# B&R Automation Studio project CleanChemi_SiteManagementSystem (part 2)

### Global.typ - Global data types
```iecst
(*Global Structrues*)
(**)
(*Raw Modbus Data*)

TYPE
	Modbus_Type : 	STRUCT
		Modbus_Alarms : Modbus_Alarm_Type;
		Modbus_Dosing : Modbus_7000_Type;
		Modbus_PeroxyMAX : Modbus_6000_Type;
	END_STRUCT;
END_TYPE

(*Raw Modbus IO*)

TYPE
	Modbus_Alarm_Type : 	STRUCT
		Block48_Int : ARRAY[0..60]OF INT;
	END_STRUCT;
	Modbus_6000_Type : 	STRUCT
		Block1_Int : ARRAY[0..124]OF INT;
		Block2_Int : ARRAY[0..248]OF USINT;
		Block3_Real : ARRAY[0..62]OF REAL;
		Block4_Real : ARRAY[0..62]OF REAL;
		Block5_Real : ARRAY[0..62]OF REAL;
	END_STRUCT;
	Modbus_7000_Type : 	STRUCT
		Block6_Int : ARRAY[0..124]OF INT;
		Block7_Int : ARRAY[0..124]OF INT;
		Block61_Int : ARRAY[0..248]OF USINT;
		Block8_Real : ARRAY[0..62]OF REAL;
		Block9_Real : ARRAY[0..62]OF REAL;
		Block10_Real : ARRAY[0..62]OF REAL;
		Block11_Real : ARRAY[0..62]OF REAL;
	END_STRUCT;
END_TYPE

(**)
(*Final Mapping Variables*)

TYPE
	Skid_type : 	STRUCT
		Pmax_Pump_101 : Pmax_Pump_101_Type;
		Pmax_Pump_101B : Pmax_Pump_101B_Type;
		Pmax_Pump_102 : Pmax_Pump_102_Type;
		Pmax_Pump_103 : Pmax_Pump_103_Type;
		Pmax_Pump_104 : Pmax_Pump_104_Type;
		BufferTank : BufferTank_Variables_Type;
		ConversionRatios : ConversionRatios_Type;
		Sensor_Variables : Sensor_Variables_Type;
		Heartbeat : Heartbeat_Type;
		Status : Status_Type;
		Alarms : Alarms_Type;
		Pmax_General_Variables : Pmax_General_Variables_Type;
		Dosing_Pump_201 : Dosing_Pump_201_Type;
		Dosing_Pump_202 : Dosing_Pump_202_Type;
		Dosing_Pump_203 : Dosing_Pump_203_Type;
		Dosing_Pump_204 : Dosing_Pump_204_Type;
		Dosing_Pump_205 : Dosing_Pump_205_Type;
		Dosing_Pump_206 : Dosing_Pump_206_Type;
		Dosing_Pump_207 : Dosing_Pump_207_Type;
		Dosing_Pump_208 : Dosing_Pump_208_Type;
		VisNum : VisNum_Type;
		VisBool : VisBool_Type;
		ErrorInfo : Skid_ErrorInfo_typ;
		tempAlarm : HA_AlarmX_Core_Buffer_typ;
		Error : BOOL;
		StateResetAlarms : UINT;
		AlarmStartupDelay : TON;
		AlarmXHistory_MpLink : MpComIdentType;
		AlarmX_MpLink : MpComIdentType;
		AlarmCfg : MpAlarmXAlarmConfigType;
		MpAlarmXConfigAlarm : MpAlarmXConfigAlarm;
		i : USINT;
		AlarmName : STRING[80];
		AlarmsInitialized : BOOL;
		Notes : Notes_Type;
		AlarmConfig : AlarmConfig_Type;
		RosterContact : RosterContact_Type;
		UserLock_LastName : STRING[80];
		UserLock_FirstName : STRING[80];
		UserLock : UINT;
	END_STRUCT;
END_TYPE

(**)
(*Alarm Text Messaging Internal CCI Roster*)

TYPE
	RosterContact_Type : 	STRUCT
		Write_Step1 : INT := 0;
		Write_Step2 : INT := 0;
		Write_Step3 : INT := 0;
		Write_Step4 : INT := 0;
		Write_Step5 : INT := 0;
		Write_Step6 : INT := 0;
		Write_Step7 : INT := 0;
		Write_Step8 : INT := 0;
		Contact1_ENABLE : BOOL;
		Contact2_ENABLE : BOOL;
		Contact3_ENABLE : BOOL;
		Contact4_ENABLE : BOOL;
		Contact5_ENABLE : BOOL;
		Contact6_ENABLE : BOOL;
		Contact7_ENABLE : BOOL;
		Contact8_ENABLE : BOOL; (*Pump 202 Visualization Enable Bit 0 = Visible  1 = Hidden*)
		Contact1 : STRING[80];
		Contact2 : STRING[80];
		Contact3 : STRING[80];
		Contact4 : STRING[80];
		Contact5 : STRING[80];
		Contact6 : STRING[80];
		Contact7 : STRING[80];
		Contact8 : STRING[80];
		Phone_Read1 : STRING[10];
		Phone_Read2 : STRING[10];
		Phone_Read3 : STRING[10];
		Phone_Read4 : STRING[10];
		Phone_Read5 : STRING[10];
		Phone_Read6 : STRING[10];
		Phone_Read7 : STRING[10];
		Phone_Read8 : STRING[10];
		Phone_Input1 : STRING[10];
		Phone_Input2 : STRING[10];
		Phone_Input3 : STRING[10];
		Phone_Input4 : STRING[10];
		Phone_Input5 : STRING[10];
		Phone_Input6 : STRING[10];
		Phone_Input7 : STRING[10];
		Phone_Input8 : STRING[10];
	END_STRUCT;
END_TYPE

(*Visualization Components*)

TYPE
	Skid_ErrorInfo_typ : 	STRUCT
		State : STRING[80];
		Text : STRING[255];
		Severity : USINT;
	END_STRUCT;
END_TYPE

(**)

TYPE
	Par_System_type : 	STRUCT
		LanguageCode : STRING[80];
	END_STRUCT;
END_TYPE

(*Retain Machine State After Power Cycle*)

TYPE
	Par_Type : 	STRUCT
		System : Par_System_type;
	END_STRUCT;
END_TYPE

(**)
(*Retain Parameter After Power Cycle*)

TYPE
	Rem_Type : 	STRUCT
		New_Member : USINT;
	END_STRUCT;
END_TYPE

(**)
(*Master Write Command *)

TYPE
	CMD_Type : 	STRUCT
		Stop : BOOL;
		Start : BOOL;
		Write_ESTOP : CMD_Write_ESTOP_Type;
		Write_UNIT_ID : CMD_Write_UNIT_ID_Type;
		Write_UNIT_ACK : CMD_Write_UNIT_ACK_Type;
		Write_P203_STP_CMD : CMD_Write_P203_STP_CMD_Type;
		Write_P203_STRT_CMD : CMD_Write_P203_STRT_CMD_Type;
		Write_P203_HOA : CMD_Write_P203_HOA_Type;
		Write_P203_PPM : CMD_Write_P203_PPM_Type;
		Write_P203_SP : CMD_Write_P203_SP_Type;
		Write_P202_STP_CMD : CMD_Write_P202_STP_CMD_Type;
		Write_P202_STRT_CMD : CMD_Write_P202_STRT_CMD_Type;
		Write_P202_HOA : CMD_Write_P202_HOA_Type;
		Write_P202_PPM : CMD_Write_P202_PPM_Type;
		Write_P202_SP : CMD_Write_P202_SP_Type;
		Write_P104_STP_CMD : CMD_Write_P104_STP_CMD_Type;
		Write_P104_STRT_CMD : CMD_Write_P104_STRT_CMD_Type;
		Write_P104_SP : CMD_Write_P104_SP_Type;
		Write_P103_STP_CMD : CMD_Write_P103_STP_CMD_Type;
		Write_P103_STRT_CMD : CMD_Write_P103_STRT_CMD_Type;
		Write_P103_SP : CMD_Write_P103_SP_Type;
		Write_P102_STP_CMD : CMD_Write_P102_STP_CMD_Type;
		Write_P102_STRT_CMD : CMD_Write_P102_STRT_CMD_Type;
		Write_P102_SP : CMD_Write_P102_SP_Type;
		Write_P101_STP_CMD : CMD_Write_P101_STP_CMD_Type;
		Write_P101_STRT_CMD : CMD_Write_P101_STRT_CMD_Type;
		Write_P101_SP : CMD_Write_P101_SP_Type;
		Write_P201_STP_CMD : CMD_Write_P201_STP_CMD_Type;
		Write_P201_STRT_CMD : CMD_Write_P201_STRT_CMD_Type;
		Write_P201_HOA : CMD_Write_P201_HOA_Type;
		Write_P201_PPM : CMD_Write_P201_PPM_Type;
		Write_P201_SP : CMD_Write_P201_SP_Type;
		Write_EFF_1 : CMD_Write_EFF_1_Type;
		Write_EFF_2 : CMD_Write_EFF_2_Type;
		Write_NAOH_TO_H2O2 : CMD_Write_NAOH_TO_H2O2_Type;
		Write_TRI_TO_H2O2 : CMD_Write_TRI_TO_H2O2_Type;
		Write_PMAX_HOA : CMD_Write_PMAX_HOA_Type;
		Write_PMAX_CONC : CMD_Write_PMAX_CONC_Type;
		Write_HP_CONC : CMD_Write_HP_CONC_Type;
		Write_NAOH_CONC : CMD_Write_NAOH_CONC_Type;
		Write_UNLOCK_CMD : CMD_Write_UNLOCK_CMD_Type;
		Write_LOCK_CMD : CMD_Write_LOCK_CMD_Type;
		Write_FI301_SIM_CMD : CMD_Write_FI301_SIM_CMD_Type;
		Write_FI301_MEA_CMD : CMD_Write_FI301_MEA_CMD_Type;
		Write_FI301_SIM : CMD_Write_FI301_SIM_Type;
		Write_FI302_SIM_CMD : CMD_Write_FI302_SIM_CMD_Type;
		Write_FI302_MEA_CMD : CMD_Write_FI302_MEA_CMD_Type;
		Write_FI302_SIM : CMD_Write_FI302_SIM_Type;
		Write_FI303_SIM_CMD : CMD_Write_FI303_SIM_CMD_Type;
		Write_FI303_MEA_CMD : CMD_Write_FI303_MEA_CMD_Type;
		Write_FI303_SIM : CMD_Write_FI303_SIM_Type;
		Write_XV101_OPEN_CMD : CMD_Write_XV101_OPEN_CMD_Type;
		Write_XV102_OPEN_CMD : CMD_Write_XV102_OPEN_CMD_Type;
		Write_XV103_OPEN_CMD : CMD_Write_XV103_OPEN_CMD_Type;
		Write_XV104_OPEN_CMD : CMD_Write_XV104_OPEN_CMD_Type;
		Write_XV201_OPEN_CMD : CMD_Write_XV201_OPEN_CMD_Type;
		Write_XV202_OPEN_CMD : CMD_Write_XV202_OPEN_CMD_Type;
		Write_XV203_OPEN_CMD : CMD_Write_XV203_OPEN_CMD_Type;
		Write_XV204_OPEN_CMD : CMD_Write_XV204_OPEN_CMD_Type;
		Write_RECALC_CMD : CMD_Write_RECALC_CMD_Type;
		Write_USERADMIN_RESET : CMD_Write_USERADMIN_RESET_Type;
		Write_TOTALIZER_RESET : CMD_Write_TOTALIZER_RESET_Type;
		Write_AS_USER : CMD_Write_AS_USER_Type;
		Write_AS_ACCESS : CMD_Write_AS_ACCESS_Type;
		Write_P204_STP_CMD : CMD_Write_P204_STP_CMD_Type;
		Write_P204_STRT_CMD : CMD_Write_P204_STRT_CMD_Type;
		Write_P204_HOA : CMD_Write_P204_HOA_Type;
		Write_P204_PPM : CMD_Write_P204_PPM_Type;
		Write_P204_SP : CMD_Write_P204_SP_Type;
		Write_FI304_SIM_CMD : CMD_Write_FI304_SIM_CMD_Type;
		Write_FI304_MEA_CMD : CMD_Write_FI304_MEA_CMD_Type;
		Write_FI304_SIM : CMD_Write_FI304_SIM_Type;
		Write_P101_AUTOCAL : CMD_Write_P101_AUTOCAL_Type;
		Write_P101_GAIN : CMD_Write_P101_GAIN_Type;
		Write_P101_STEPADJ : CMD_Write_P101_STEPADJ_Type;
		Write_P101_TOTALADJ : CMD_Write_P101_TOTALADJ_Type;
		Write_P102_AUTOFLO_ADPT : CMD_Write_P102_AUTOFLO_ADPT_Type;
		Write_P102_AUTOCAL : CMD_Write_P102_AUTOCAL_Type;
		Write_P102_GAIN : CMD_Write_P102_GAIN_Type;
		Write_P102_STEPADJ : CMD_Write_P102_STEPADJ_Type;
		Write_P102_TOTALADJ : CMD_Write_P102_TOTALADJ_Type;
		Write_P103_AUTOFLO_ADPT : CMD_Write_P103_AUTOFLO_ADPT_Type;
		Write_P103_AUTOCAL : CMD_Write_P103_AUTOCAL_Type;
		Write_P103_GAIN : CMD_Write_P103_GAIN_Type;
		Write_P103_STEPADJ : CMD_Write_P103_STEPADJ_Type;
		Write_P103_TOTALADJ : CMD_Write_P103_TOTALADJ_Type;
		Write_P104_AUTOFLO_ADPT : CMD_Write_P104_AUTOFLO_ADPT_Type;
		Write_P104_AUTOCAL : CMD_Write_P104_AUTOCAL_Type;
		Write_P104_AUTOCAL_PV : CMD_Write_P104_AUTOCAL_PV_Type;
		Write_P104_GAIN : CMD_Write_P104_GAIN_Type;
		Write_P104_STEPADJ : CMD_Write_P104_STEPADJ_Type;
		Write_P104_TOTALADJ : CMD_Write_P104_TOTALADJ_Type;
		Write_P201_AUTOFLO_ADPT : CMD_Write_P201_AUTOFLO_ADPT_Type;
		Write_P201_AUTOCAL : CMD_Write_P201_AUTOCAL_Type;
		Write_P201_AUTOCAL_PV : CMD_Write_P201_AUTOCAL_PV_Type;
		Write_P201_GAIN : CMD_Write_P201_GAIN_Type;
		Write_P201_STEPADJ : CMD_Write_P201_STEPADJ_Type;
		Write_P201_TOTALADJ : CMD_Write_P201_TOTALADJ_Type;
		Write_P202_AUTOFLO_ADPT : CMD_Write_P202_AUTOFLO_ADPT_Type;
		Write_P202_AUTOCAL : CMD_Write_P202_AUTOCAL_Type;
		Write_P202_AUTOCAL_PV : CMD_Write_P202_AUTOCAL_PV_Type;
		Write_P202_GAIN : CMD_Write_P202_GAIN_Type;
		Write_P202_STEPADJ : CMD_Write_P202_STEPADJ_Type;
		Write_P202_TOTALADJ : CMD_Write_P202_TOTALADJ_Type;
		Write_P203_AUTOFLO_ADPT : CMD_Write_P203_AUTOFLO_ADPT_Type;
		Write_P203_AUTOCAL : CMD_Write_P203_AUTOCAL_Type;
		Write_P203_AUTOCAL_PV : CMD_Write_P203_AUTOCAL_PV_Type;
		Write_P203_GAIN : CMD_Write_P203_GAIN_Type;
		Write_P203_STEPADJ : CMD_Write_P203_STEPADJ_Type;
		Write_P203_TOTALADJ : CMD_Write_P203_TOTALADJ_Type;
		Write_P204_AUTOFLO_ADPT : CMD_Write_P204_AUTOFLO_ADPT_Type;
		Write_P204_AUTOCAL : CMD_Write_P204_AUTOCAL_Type;
		Write_P204_AUTOCAL_PV : CMD_Write_P204_AUTOCAL_PV_Type;
		Write_P204_GAIN : CMD_Write_P204_GAIN_Type;
		Write_P204_STEPADJ : CMD_Write_P204_STEPADJ_Type;
		Write_P204_TOTALADJ : CMD_Write_P204_TOTALADJ_Type;
		Write_PHONE_INPUT1 : CMD_Write_PHONE_INPUT1_Type;
		Write_PHONE_INPUT2 : CMD_Write_PHONE_INPUT2_Type;
		Write_PHONE_INPUT3 : CMD_Write_PHONE_INPUT3_Type;
		Write_PHONE_INPUT4 : CMD_Write_PHONE_INPUT4_Type;
		Write_PHONE_INPUT5 : CMD_Write_PHONE_INPUT5_Type;
		Write_PHONE_INPUT6 : CMD_Write_PHONE_INPUT6_Type;
		Write_PHONE_INPUT7 : CMD_Write_PHONE_INPUT7_Type;
		Write_PHONE_INPUT8 : CMD_Write_PHONE_INPUT8_Type;
		Write_ENABLE_ROSTER1 : CMD_Write_ENABLE_ROSTER1_Type;
		Write_ENABLE_ROSTER2 : CMD_Write_ENABLE_ROSTER2_Type;
		Write_ENABLE_ROSTER3 : CMD_Write_ENABLE_ROSTER3_Type;
		Write_ENABLE_ROSTER4 : CMD_Write_ENABLE_ROSTER4_Type;
		Write_ENABLE_ROSTER5 : CMD_Write_ENABLE_ROSTER5_Type;
		Write_ENABLE_ROSTER6 : CMD_Write_ENABLE_ROSTER6_Type;
		Write_ENABLE_ROSTER7 : CMD_Write_ENABLE_ROSTER7_Type;
		Write_ENABLE_ROSTER8 : CMD_Write_ENABLE_ROSTER8_Type;
		Write_AC_ALARM_ENABLE : CMD_Write_AC_ALARM_ENABLE_Type;
		Write_AC_TXT_ENABLE : CMD_Write_AC_TXT_ENABLE_Type;
		Write_AC_ACTION : CMD_Write_AC_ACTION_Type;
		Write_AC_DELAY : CMD_Write_AC_DELAY_Type;
		Write_AC_OFFSET : CMD_Write_AC_OFFSET_Type;
		Write_AC_THRESHOLD : CMD_Write_AC_THRESHOLD_Type;
	END_STRUCT;
END_TYPE

(**)
(*Misc. Write Commands*)

TYPE
	CMD_Write_ESTOP_Type : 	STRUCT
		wESTOP : UINT := 1;
		Send : BOOL;
	END_STRUCT;
	CMD_Write_UNIT_ACK_Type : 	STRUCT
		wUNIT_ACK : UINT := 1;
	END_STRUCT;
	CMD_Write_AS_ACCESS_Type : 	STRUCT
		Send : BOOL;
		wAS_ACCESS : UINT := 1;
	END_STRUCT;
	CMD_Write_AS_USER_Type : 	STRUCT
		Send : BOOL;
		wAS_USER : UINT := 1;
	END_STRUCT;
	CMD_Write_RECALC_CMD_Type : 	STRUCT
		Send : BOOL;
		wRECALC_CMD : UINT := 1;
	END_STRUCT;
	CMD_Write_USERADMIN_RESET_Type : 	STRUCT
		Send : BOOL;
		wUSERADMIN_RESET : UINT := 1111;
	END_STRUCT;
	CMD_Write_TOTALIZER_RESET_Type : 	STRUCT
		Send : BOOL;
		wTOTALIZER_RESET : UINT := 1;
	END_STRUCT;
	CMD_Write_UNLOCK_CMD_Type : 	STRUCT
		Send : BOOL;
		wUNLOCK_CMD : UINT := 1;
	END_STRUCT;
	CMD_Write_LOCK_CMD_Type : 	STRUCT
		Send : BOOL;
		wLOCK_CMD : UINT := 1;
	END_STRUCT;
	CMD_Write_EFF_1_Type : 	STRUCT
		Send : BOOL;
		wEFF_1 : REAL;
		wEFF_1_SWAPPED : REAL;
	END_STRUCT;
	CMD_Write_EFF_2_Type : 	STRUCT
		Send : BOOL;
		wEFF_2 : REAL;
		wEFF_2_SWAPPED : REAL;
	END_STRUCT;
	CMD_Write_NAOH_TO_H2O2_Type : 	STRUCT
		Send : BOOL;
		wNAOH_TO_H2O2 : REAL;
		wNAOH_TO_H2O2_SWAPPED : REAL;
	END_STRUCT;
	CMD_Write_TRI_TO_H2O2_Type : 	STRUCT
		Send : BOOL;
		wTRI_TO_H2O2 : REAL;
		wTRI_TO_H2O2_SWAPPED : REAL;
	END_STRUCT;
	CMD_Write_PMAX_HOA_Type : 	STRUCT
		Send : BOOL;
		wPMAX_HOA : UINT;
		Cancel : BOOL;
		wPMAX_HOA_String : STRING[80];
	END_STRUCT;
	CMD_Write_PMAX_CONC_Type : 	STRUCT
		Send : BOOL;
		wPMAX_CONC : REAL;
		wPMAX_CONC_SWAPPED : REAL;
	END_STRUCT;
	CMD_Write_HP_CONC_Type : 	STRUCT
		Send : BOOL;
		wHP_CONC : REAL;
		wHP_CONC_SWAPPED : REAL;
	END_STRUCT;
	CMD_Write_NAOH_CONC_Type : 	STRUCT
		Send : BOOL;
		wNAOH_CONC : REAL;
		wNAOH_CONC_SWAPPED : REAL;
	END_STRUCT;
END_TYPE

(*P101 Write Commands*)

TYPE
	CMD_Write_P101_STP_CMD_Type : 	STRUCT
		Send : BOOL;
		wP101_STP_CMD : UINT := 1;
	END_STRUCT;
	CMD_Write_P101_STRT_CMD_Type : 	STRUCT
		Send : BOOL;
		wP101_STRT_CMD : UINT := 1;
	END_STRUCT;
	CMD_Write_P101_SP_Type : 	STRUCT
		Send : BOOL;
		wP101_SP : REAL;
		wP101_SP_SWAPPED : REAL;
	END_STRUCT;
	CMD_Write_P101_AUTOCAL_Type : 	STRUCT
		Send : BOOL;
		wP101_AUTOCAL : UINT := 1;
	END_STRUCT;
	CMD_Write_P101_GAIN_Type : 	STRUCT
		Send : BOOL;
		wP101_GAIN : REAL;
		wP101_GAIN_SWAPPED : REAL;
	END_STRUCT;
	CMD_Write_P101_STEPADJ_Type : 	STRUCT
		Send : BOOL;
		wP101_STEPADJ : REAL;
		wP101_STEPADJ_SWAPPED : REAL;
	END_STRUCT;
	CMD_Write_P101_TOTALADJ_Type : 	STRUCT
		Send : BOOL;
		wP101_TOTALADJ : REAL;
		wP101_TOTALADJ_SWAPPED : REAL;
	END_STRUCT;
END_TYPE

(*P102 Write Commands*)

TYPE
	CMD_Write_P102_STP_CMD_Type : 	STRUCT
		Send : BOOL;
		wP102_STP_CMD : UINT := 1;
	END_STRUCT;
	CMD_Write_P102_STRT_CMD_Type : 	STRUCT
		Send : BOOL;
		wP102_STRT_CMD : UINT := 1;
	END_STRUCT;
	CMD_Write_P102_SP_Type : 	STRUCT
		Send : BOOL;
		wP102_SP : REAL;
		wP102_SP_SWAPPED : REAL;
	END_STRUCT;
	CMD_Write_P102_AUTOFLO_ADPT_Type : 	STRUCT
		Send : BOOL;
		wP102_P102_AUTOFLO_ADPT : UINT := 1;
	END_STRUCT;
	CMD_Write_P102_AUTOCAL_Type : 	STRUCT
		Send : BOOL;
		wP102_AUTOCAL : UINT := 1;
	END_STRUCT;
	CMD_Write_P102_GAIN_Type : 	STRUCT
		Send : BOOL;
		wP102_GAIN : REAL;
		wP102_GAIN_SWAPPED : REAL;
	END_STRUCT;
	CMD_Write_P102_STEPADJ_Type : 	STRUCT
		Send : BOOL;
		wP102_STEPADJ : REAL;
		wP102_STEPADJ_SWAPPED : REAL;
	END_STRUCT;
	CMD_Write_P102_TOTALADJ_Type : 	STRUCT
		Send : BOOL;
		wP102_TOTALADJ : REAL;
		wP102_TOTALADJ_SWAPPED : REAL;
	END_STRUCT;
END_TYPE

(*P103 Write Commands*)

TYPE
	CMD_Write_P103_STP_CMD_Type : 	STRUCT
		Send : BOOL;
		wP103_STP_CMD : UINT := 1;
	END_STRUCT;
	CMD_Write_P103_STRT_CMD_Type : 	STRUCT
		Send : BOOL;
		wP103_STRT_CMD : UINT := 1;
	END_STRUCT;
	CMD_Write_P103_SP_Type : 	STRUCT
		Send : BOOL;
		wP103_SP : REAL;
		wP103_SP_SWAPPED : REAL;
	END_STRUCT;
	CMD_Write_P103_AUTOFLO_ADPT_Type : 	STRUCT
		Send : BOOL;
		wP103_P103_AUTOFLO_ADPT : UINT := 1;
	END_STRUCT;
	CMD_Write_P103_AUTOCAL_Type : 	STRUCT
		Send : BOOL;
		wP103_AUTOCAL : UINT := 1;
	END_STRUCT;
	CMD_Write_P103_GAIN_Type : 	STRUCT
		Send : BOOL;
		wP103_GAIN : REAL;
		wP103_GAIN_SWAPPED : REAL;
	END_STRUCT;
	CMD_Write_P103_STEPADJ_Type : 	STRUCT
		Send : BOOL;
		wP103_STEPADJ : REAL;
		wP103_STEPADJ_SWAPPED : REAL;
	END_STRUCT;
	CMD_Write_P103_TOTALADJ_Type : 	STRUCT
		Send : BOOL;
		wP103_TOTALADJ : REAL;
		wP103_TOTALADJ_SWAPPED : REAL;
	END_STRUCT;
END_TYPE

(*P104 Write Commands*)

TYPE
	CMD_Write_P104_STP_CMD_Type : 	STRUCT
		Send : BOOL;
		wP104_STP_CMD : UINT := 1;
	END_STRUCT;
	CMD_Write_P104_STRT_CMD_Type : 	STRUCT
		Send : BOOL;
		wP104_STRT_CMD : UINT := 1;
	END_STRUCT;
	CMD_Write_P104_SP_Type : 	STRUCT
		Send : BOOL;
		wP104_SP : REAL;
		wP104_SP_SWAPPED : REAL;
	END_STRUCT;
	CMD_Write_P104_AUTOFLO_ADPT_Type : 	STRUCT
		Send : BOOL;
		wP104_P104_AUTOFLO_ADPT : UINT := 1;
	END_STRUCT;
	CMD_Write_P104_AUTOCAL_Type : 	STRUCT
		Send : BOOL;
		wP104_AUTOCAL : UINT := 1;
	END_STRUCT;
	CMD_Write_P104_AUTOCAL_PV_Type : 	STRUCT
		Send : BOOL;
		wP104_AUTOCAL_PV : UINT := 1;
	END_STRUCT;
	CMD_Write_P104_GAIN_Type : 	STRUCT
		Send : BOOL;
		wP104_GAIN : REAL;
		wP104_GAIN_SWAPPED : REAL;
	END_STRUCT;
	CMD_Write_P104_STEPADJ_Type : 	STRUCT
		Send : BOOL;
		wP104_STEPADJ : REAL;
		wP104_STEPADJ_SWAPPED : REAL;
	END_STRUCT;
	CMD_Write_P104_TOTALADJ_Type : 	STRUCT
		Send : BOOL;
		wP104_TOTALADJ : REAL;
		wP104_TOTALADJ_SWAPPED : REAL;
	END_STRUCT;
END_TYPE

(*P201 Write Commands*)

TYPE
	CMD_Write_P201_STP_CMD_Type : 	STRUCT
		Send : BOOL;
		wP201_STP_CMD : UINT := 1;
	END_STRUCT;
	CMD_Write_P201_STRT_CMD_Type : 	STRUCT
		Send : BOOL;
		wP201_STRT_CMD : UINT := 1;
	END_STRUCT;
	CMD_Write_P201_SP_Type : 	STRUCT
		Send : BOOL;
		wP201_SP : REAL;
		wP201_SP_SWAPPED : REAL;
	END_STRUCT;
	CMD_Write_P201_PPM_Type : 	STRUCT
		Send : BOOL;
		wP201_PPM : REAL;
		wP201_PPM_SWAPPED : REAL;
	END_STRUCT;
	CMD_Write_P201_HOA_Type : 	STRUCT
		Cancel : BOOL;
		Send : BOOL;
		wP201_HOA_String : STRING[80];
		wP201_HOA : UINT;
	END_STRUCT;
	CMD_Write_P201_AUTOFLO_ADPT_Type : 	STRUCT
		Send : BOOL;
		wP201_P201_AUTOFLO_ADPT : UINT := 1;
	END_STRUCT;
	CMD_Write_P201_AUTOCAL_Type : 	STRUCT
		Send : BOOL;
		wP201_AUTOCAL : UINT := 1;
	END_STRUCT;
	CMD_Write_P201_AUTOCAL_PV_Type : 	STRUCT
		Send : BOOL;
		wP201_AUTOCAL_PV : UINT := 1;
	END_STRUCT;
	CMD_Write_P201_GAIN_Type : 	STRUCT
		Send : BOOL;
		wP201_GAIN : REAL;
		wP201_GAIN_SWAPPED : REAL;
	END_STRUCT;
	CMD_Write_P201_STEPADJ_Type : 	STRUCT
		Send : BOOL;
		wP201_STEPADJ : REAL;
		wP201_STEPADJ_SWAPPED : REAL;
	END_STRUCT;
	CMD_Write_P201_TOTALADJ_Type : 	STRUCT
		Send : BOOL;
		wP201_TOTALADJ : REAL;
		wP201_TOTALADJ_SWAPPED : REAL;
	END_STRUCT;
END_TYPE

(*P202 Write Commands*)

TYPE
	CMD_Write_P202_STP_CMD_Type : 	STRUCT
		Send : BOOL;
		wP202_STP_CMD : UINT := 1;
	END_STRUCT;
	CMD_Write_P202_STRT_CMD_Type : 	STRUCT
		Send : BOOL;
		wP202_STRT_CMD : UINT := 1;
	END_STRUCT;
	CMD_Write_P202_SP_Type : 	STRUCT
		Send : BOOL;
		wP202_SP : REAL;
		wP202_SP_SWAPPED : REAL;
	END_STRUCT;
	CMD_Write_P202_PPM_Type : 	STRUCT
		Send : BOOL;
		wP202_PPM : REAL;
		wP202_PPM_SWAPPED : REAL;
	END_STRUCT;
	CMD_Write_P202_HOA_Type : 	STRUCT
		Cancel : BOOL;
		Send : BOOL;
		wP202_HOA_String : STRING[80];
		wP202_HOA : UINT;
	END_STRUCT;
	CMD_Write_P202_AUTOFLO_ADPT_Type : 	STRUCT
		Send : BOOL;
		wP202_P202_AUTOFLO_ADPT : UINT := 1;
	END_STRUCT;
	CMD_Write_P202_AUTOCAL_Type : 	STRUCT
		Send : BOOL;
		wP202_AUTOCAL : UINT := 1;
	END_STRUCT;
	CMD_Write_P202_AUTOCAL_PV_Type : 	STRUCT
		Send : BOOL;
		wP202_AUTOCAL_PV : UINT := 1;
	END_STRUCT;
	CMD_Write_P202_GAIN_Type : 	STRUCT
		Send : BOOL;
		wP202_GAIN : REAL;
		wP202_GAIN_SWAPPED : REAL;
	END_STRUCT;
	CMD_Write_P202_STEPADJ_Type : 	STRUCT
		Send : BOOL;
		wP202_STEPADJ : REAL;
		wP202_STEPADJ_SWAPPED : REAL;
	END_STRUCT;
	CMD_Write_P202_TOTALADJ_Type : 	STRUCT
		Send : BOOL;
		wP202_TOTALADJ : REAL;
		wP202_TOTALADJ_SWAPPED : REAL;
	END_STRUCT;
END_TYPE

(*P203 Write Commands*)

TYPE
	CMD_Write_P203_STP_CMD_Type : 	STRUCT
		Send : BOOL;
		wP203_STP_CMD : UINT := 1;
	END_STRUCT;
	CMD_Write_P203_STRT_CMD_Type : 	STRUCT
		Send : BOOL;
		wP203_STRT_CMD : UINT := 1;
	END_STRUCT;
	CMD_Write_P203_SP_Type : 	STRUCT
		Send : BOOL;
		wP203_SP : REAL;
		wP203_SP_SWAPPED : REAL;
	END_STRUCT;
	CMD_Write_P203_PPM_Type : 	STRUCT
		Send : BOOL;
		wP203_PPM : REAL;
		wP203_PPM_SWAPPED : REAL;
	END_STRUCT;
	CMD_Write_P203_HOA_Type : 	STRUCT
		Send : BOOL;
		wP203_HOA : UINT;
		Cancel : BOOL;
		wP203_HOA_String : STRING[80];
	END_STRUCT;
	CMD_Write_P203_AUTOFLO_ADPT_Type : 	STRUCT
		Send : BOOL;
		wP203_P203_AUTOFLO_ADPT : UINT := 1;
	END_STRUCT;
	CMD_Write_P203_AUTOCAL_Type : 	STRUCT
		Send : BOOL;
		wP203_AUTOCAL : UINT := 1;
	END_STRUCT;
	CMD_Write_P203_AUTOCAL_PV_Type : 	STRUCT
		Send : BOOL;
		wP203_AUTOCAL_PV : UINT := 1;
	END_STRUCT;
	CMD_Write_P203_GAIN_Type : 	STRUCT
		Send : BOOL;
		wP203_GAIN : REAL;
		wP203_GAIN_SWAPPED : REAL;
	END_STRUCT;
	CMD_Write_P203_STEPADJ_Type : 	STRUCT
		Send : BOOL;
		wP203_STEPADJ : REAL;
		wP203_STEPADJ_SWAPPED : REAL;
	END_STRUCT;
	CMD_Write_P203_TOTALADJ_Type : 	STRUCT
		Send : BOOL;
		wP203_TOTALADJ : REAL;
		wP203_TOTALADJ_SWAPPED : REAL;
	END_STRUCT;
END_TYPE

(*P204 Write Commands*)

TYPE
	CMD_Write_P204_STP_CMD_Type : 	STRUCT
		Send : BOOL;
		wP204_STP_CMD : UINT := 1;
	END_STRUCT;
	CMD_Write_P204_STRT_CMD_Type : 	STRUCT
		Send : BOOL;
		wP204_STRT_CMD : UINT := 1;
	END_STRUCT;
	CMD_Write_P204_SP_Type : 	STRUCT
		Send : BOOL;
		wP204_SP : REAL;
		wP204_SP_SWAPPED : REAL;
	END_STRUCT;
	CMD_Write_P204_PPM_Type : 	STRUCT
		Send : BOOL;
		wP204_PPM : REAL;
		wP204_PPM_SWAPPED : REAL;
	END_STRUCT;
	CMD_Write_P204_HOA_Type : 	STRUCT
		Send : BOOL;
		wP204_HOA : UINT;
		Cancel : BOOL;
		wP204_HOA_String : STRING[80];
	END_STRUCT;
	CMD_Write_P204_AUTOFLO_ADPT_Type : 	STRUCT
		Send : BOOL;
		wP204_P204_AUTOFLO_ADPT : UINT := 1;
	END_STRUCT;
	CMD_Write_P204_AUTOCAL_Type : 	STRUCT
		Send : BOOL;
		wP204_AUTOCAL : UINT := 1;
	END_STRUCT;
	CMD_Write_P204_AUTOCAL_PV_Type : 	STRUCT
		Send : BOOL;
		wP204_AUTOCAL_PV : UINT := 1;
	END_STRUCT;
	CMD_Write_P204_GAIN_Type : 	STRUCT
		Send : BOOL;
		wP204_GAIN : REAL;
		wP204_GAIN_SWAPPED : REAL;
	END_STRUCT;
	CMD_Write_P204_STEPADJ_Type : 	STRUCT
		Send : BOOL;
		wP204_STEPADJ : REAL;
		wP204_STEPADJ_SWAPPED : REAL;
	END_STRUCT;
	CMD_Write_P204_TOTALADJ_Type : 	STRUCT
		Send : BOOL;
		wP204_TOTALADJ : REAL;
		wP204_TOTALADJ_SWAPPED : REAL;
	END_STRUCT;
END_TYPE

(*UID Write Command*)

TYPE
	CMD_Write_UNIT_ID_Type : 	STRUCT
		Send : BOOL;
		wUNIT_ID : UINT;
	END_STRUCT;
END_TYPE

(*FI301 Write Commands*)

TYPE
	CMD_Write_FI301_SIM_CMD_Type : 	STRUCT
		Send : BOOL;
		wFI301_SIM_CMD : UINT := 1;
	END_STRUCT;
	CMD_Write_FI301_MEA_CMD_Type : 	STRUCT
		Send : BOOL;
		wFI301_MEA_CMD : UINT := 1;
	END_STRUCT;
	CMD_Write_FI301_SIM_Type : 	STRUCT
		Send : BOOL;
		wFI301_SIM : REAL;
		wFI301_SIM_SWAPPED : REAL;
	END_STRUCT;
END_TYPE

(*FI302 Write Commands*)

TYPE
	CMD_Write_FI302_SIM_CMD_Type : 	STRUCT
		Send : BOOL;
		wFI302_SIM_CMD : UINT := 1;
	END_STRUCT;
	CMD_Write_FI302_MEA_CMD_Type : 	STRUCT
		Send : BOOL;
		wFI302_MEA_CMD : UINT := 1;
	END_STRUCT;
	CMD_Write_FI302_SIM_Type : 	STRUCT
		Send : BOOL;
		wFI302_SIM : REAL;
		wFI302_SIM_SWAPPED : REAL;
	END_STRUCT;
END_TYPE

(*FI303 Write Commands*)

TYPE
	CMD_Write_FI303_SIM_CMD_Type : 	STRUCT
		Send : BOOL;
		wFI303_SIM_CMD : UINT := 1;
	END_STRUCT;
	CMD_Write_FI303_MEA_CMD_Type : 	STRUCT
		Send : BOOL;
		wFI303_MEA_CMD : UINT := 1;
	END_STRUCT;
	CMD_Write_FI303_SIM_Type : 	STRUCT
		Send : BOOL;
		wFI303_SIM : REAL;
		wFI303_SIM_SWAPPED : REAL;
	END_STRUCT;
END_TYPE

(*FI304 Write Commands*)

TYPE
	CMD_Write_FI304_SIM_CMD_Type : 	STRUCT
		Send : BOOL;
		wFI304_SIM_CMD : UINT := 1;
	END_STRUCT;
	CMD_Write_FI304_MEA_CMD_Type : 	STRUCT
		Send : BOOL;
		wFI304_MEA_CMD : UINT := 1;
	END_STRUCT;
	CMD_Write_FI304_SIM_Type : 	STRUCT
		Send : BOOL;
		wFI304_SIM : REAL;
		wFI304_SIM_SWAPPED : REAL;
	END_STRUCT;
END_TYPE

(*XV101 Solenoid Commands*)

TYPE
	CMD_Write_XV101_OPEN_CMD_Type : 	STRUCT
		Send : BOOL;
		wXV101_OPEN_CMD : UINT := 1;
	END_STRUCT;
END_TYPE

(*XV102 Solenoid Commands*)

TYPE
	CMD_Write_XV102_OPEN_CMD_Type : 	STRUCT
		Send : BOOL;
		wXV102_OPEN_CMD : UINT := 1;
	END_STRUCT;
END_TYPE

(*XV103 Solenoid Commands*)

TYPE
	CMD_Write_XV103_OPEN_CMD_Type : 	STRUCT
		Send : BOOL;
		wXV103_OPEN_CMD : UINT := 1;
	END_STRUCT;
END_TYPE

(*XV104 Solenoid Commands*)

TYPE
	CMD_Write_XV104_OPEN_CMD_Type : 	STRUCT
		Send : BOOL;
		wXV104_OPEN_CMD : UINT := 1;
	END_STRUCT;
END_TYPE

(*XV201 Solenoid Commands*)

TYPE
	CMD_Write_XV201_OPEN_CMD_Type : 	STRUCT
		Send : BOOL;
		wXV201_OPEN_CMD : UINT := 1;
	END_STRUCT;
END_TYPE

(*XV202 Solenoid Commands*)

TYPE
	CMD_Write_XV202_OPEN_CMD_Type : 	STRUCT
		Send : BOOL;
		wXV202_OPEN_CMD : UINT := 1;
	END_STRUCT;
END_TYPE

(*XV203 Solenoid Commands*)

TYPE
	CMD_Write_XV203_OPEN_CMD_Type : 	STRUCT
		Send : BOOL;
		wXV203_OPEN_CMD : UINT := 1;
	END_STRUCT;
END_TYPE

(*XV204 Solenoid Commands*)

TYPE
	CMD_Write_XV204_OPEN_CMD_Type : 	STRUCT
		Send : BOOL;
		wXV204_OPEN_CMD : UINT := 1;
	END_STRUCT;
END_TYPE

(*Roster Write Commands*)

TYPE
	CMD_Write_PHONE_INPUT1_Type : 	STRUCT
		Send : BOOL;
		wPHONE_INPUT1_ARRAY : ARRAY[0..4]OF UINT;
	END_STRUCT;
	CMD_Write_ENABLE_ROSTER1_Type : 	STRUCT
		Send : BOOL;
		wENABLE_ROSTER1 : UINT := 0;
	END_STRUCT;
	CMD_Write_PHONE_INPUT2_Type : 	STRUCT
		Send : BOOL;
		wPHONE_INPUT2_ARRAY : ARRAY[0..4]OF UINT;
	END_STRUCT;
	CMD_Write_ENABLE_ROSTER2_Type : 	STRUCT
		Send : BOOL;
		wENABLE_ROSTER2 : UINT := 0;
	END_STRUCT;
	CMD_Write_PHONE_INPUT3_Type : 	STRUCT
		Send : BOOL;
		wPHONE_INPUT3_ARRAY : ARRAY[0..4]OF UINT;
	END_STRUCT;
	CMD_Write_ENABLE_ROSTER3_Type : 	STRUCT
		Send : BOOL;
		wENABLE_ROSTER3 : UINT := 0;
	END_STRUCT;
	CMD_Write_PHONE_INPUT4_Type : 	STRUCT
		Send : BOOL;
		wPHONE_INPUT4_ARRAY : ARRAY[0..4]OF UINT;
	END_STRUCT;
	CMD_Write_ENABLE_ROSTER4_Type : 	STRUCT
		Send : BOOL;
		wENABLE_ROSTER4 : UINT := 0;
	END_STRUCT;
	CMD_Write_PHONE_INPUT5_Type : 	STRUCT
		Send : BOOL;
		wPHONE_INPUT5_ARRAY : ARRAY[0..4]OF UINT;
	END_STRUCT;
	CMD_Write_ENABLE_ROSTER5_Type : 	STRUCT
		Send : BOOL;
		wENABLE_ROSTER5 : UINT := 0;
	END_STRUCT;
	CMD_Write_PHONE_INPUT6_Type : 	STRUCT
		Send : BOOL;
		wPHONE_INPUT6_ARRAY : ARRAY[0..4]OF UINT;
	END_STRUCT;
	CMD_Write_ENABLE_ROSTER6_Type : 	STRUCT
		Send : BOOL;
		wENABLE_ROSTER6 : UINT := 0;
	END_STRUCT;
	CMD_Write_PHONE_INPUT7_Type : 	STRUCT
		Send : BOOL;
		wPHONE_INPUT7_ARRAY : ARRAY[0..4]OF UINT;
	END_STRUCT;
	CMD_Write_ENABLE_ROSTER7_Type : 	STRUCT
		Send : BOOL;
		wENABLE_ROSTER7 : UINT := 0;
	END_STRUCT;
	CMD_Write_PHONE_INPUT8_Type : 	STRUCT
		Send : BOOL;
		wPHONE_INPUT8_ARRAY : ARRAY[0..4]OF UINT;
	END_STRUCT;
	CMD_Write_ENABLE_ROSTER8_Type : 	STRUCT
		Send : BOOL;
		wENABLE_ROSTER8 : UINT := 0;
	END_STRUCT;
END_TYPE

(*Alarm Configuration Write Commands*)

TYPE
	CMD_Write_AC_ALARM_ENABLE_Type : 	STRUCT
		Send : BOOL;
		wAC_ALARM_ENABLE : UINT := 0;
	END_STRUCT;
	CMD_Write_AC_TXT_ENABLE_Type : 	STRUCT
		Send : BOOL;
		wAC_TXT_ENABLE : UINT := 0;
	END_STRUCT;
	CMD_Write_AC_ACTION_Type : 	STRUCT
		Send : BOOL;
		wAC_ACTION : UINT := 0;
	END_STRUCT;
	CMD_Write_AC_DELAY_Type : 	STRUCT
		Send : BOOL;
		wAC_DELAY : UDINT := 0;
	END_STRUCT;
	CMD_Write_AC_OFFSET_Type : 	STRUCT
		Send : BOOL;
		wAC_OFFSET : UINT := 0;
	END_STRUCT;
	CMD_Write_AC_THRESHOLD_Type : 	STRUCT
		Send : BOOL;
		wAC_THRESHOLD : REAL;
		wAC_THRESHOLD_SWAPPED : REAL;
	END_STRUCT;
END_TYPE

(**)

TYPE
	Vis_Type : 	STRUCT
		Pumps : USINT;
		Main : Vis_Main_Type;
		Global : Vis_Global;
		Alarms_HR : ARRAY[0..MAX_SKIDS_HR]OF Vis_Alarms_Type;
		Alarms_LR : ARRAY[0..MAX_SKIDS_LR]OF Vis_Alarms_Type;
		Alarms_Global : Vis_Alarms_Type;
		Process : Vis_Process_Type;
	END_STRUCT;
	Vis_Global : 	STRUCT
		ClientInfo : ARRAY[0..MAX_CLIENTS]OF Vis_Global_ClientInfo;
		ErrorReset : BOOL;
	END_STRUCT;
	Vis_Global_ClientInfo : 	STRUCT
		LoginFailed : BOOL;
		LogoutSuccess : BOOL;
		LoginSuccess : BOOL;
		LogoutRequest : BOOL;
		LoginRequest : BOOL;
		Password : STRING[80];
		User : STRING[80];
		SelectedSkidIdx : USINT;
		UserID : STRING[80];
		IsValid : BOOL;
		LoginBypass : BOOL;
		LoginErrorInfo : STRING[80];
		SelectedAlrm_UnitID : STRING[80];
		SelectedAlrm_Skid : STRING[80];
		GoToSkid : BOOL;
		SelectedAlrmIndx_Temp : UINT;
		SelectedAlrmIndx : UINT;
		API_FIRST_NAME : STRING[80];
		API_LAST_NAME : STRING[80];
		API_ID : UINT;
	END_STRUCT;
	Vis_Alarms_Type : 	STRUCT
		Active : Vis_Alarms_Active_typ;
		History : Vis_Alarms_History_typ;
	END_STRUCT;
	Vis_Alarms_Active_typ : 	STRUCT
		UIConnect : MpAlarmXListUIConnectType;
		Reset : BOOL;
		PageDown : BOOL;
		PageUp : BOOL;
		SelectedIndex_Temp : UINT;
		SelectedIndex : UINT;
		TableConfig : STRING[255];
		TempINT : INT;
		TempSTRING : STRING[30];
		Enable : BOOL;
		Visable : BOOL;
		AckAll : BOOL;
	END_STRUCT;
	Vis_Alarms_History_typ : 	STRUCT
		UIConnect : MpAlarmXHistoryUIConnectType;
		State : ARRAY[0..49]OF UINT;
		Clear : BOOL;
		PageDown : BOOL;
		PageUp : BOOL;
		Export : BOOL;
		SelectedIndex : UINT;
		TableConfig : STRING[255];
		TempINT : INT;
		TempSTRING : STRING[30];
	END_STRUCT;
	Vis_Main_Internal_Type : 	STRUCT
		IP_WSTRING_Temp : WSTRING[80];
		SkidAlarmName : STRING[80];
	END_STRUCT;
	Vis_Main_Out_Type : 	STRUCT
		IPAddressDataProv_HR : ARRAY[0..MAX_SKIDS_HR]OF WSTRING[80];
		IPAddressDataProv_LR : ARRAY[0..MAX_SKIDS_LR]OF WSTRING[80];
		DialogOpen : BOOL;
		SkidIPAddress_LR : ARRAY[0..MAX_SKIDS_LR]OF STRING[20];
		SkidIPAddress_HR : ARRAY[0..MAX_SKIDS_HR]OF STRING[20];
	END_STRUCT;
	Vis_Main_In_Type : 	STRUCT
		SelectedSkidSessionVar : INT;
		AckAllAlarms_Skid_HR : ARRAY[0..100]OF BOOL;
		AckAllAlarms_Skid_LR : ARRAY[0..100]OF BOOL;
	END_STRUCT;
	Vis_Process_Internal_Type : 	STRUCT
		In : Vis_Main_In_Type;
		Internal : Vis_Main_Internal_Type;
		Out : Vis_Main_Out_Type;
	END_STRUCT;
	Vis_Process_Out_ST_Type : 	STRUCT
		PI101_Indicator : STRING[80];
		PI101_Gauge : REAL;
		CD101_Indicator : STRING[80];
		CD101_Gauge : REAL;
		CD102_Indicator : STRING[80];
		CD102_Gauge : REAL;
		GEN_Indicator : STRING[80];
		UNIT_Indicator : STRING[80];
		P201_Indicator : STRING[80];
		P202_Indicator : STRING[80];
		P203_Indicator : STRING[80];
		FI_PlantFlowCombined : REAL;
		UnitNumber : STRING[80];
	END_STRUCT;
	Vis_Process_Out_Type : 	STRUCT
		SummaryTiles : ARRAY[0..MAX_SKIDS_LR]OF Vis_Process_Out_ST_Type;
	END_STRUCT;
	Vis_Process_In_Type : 	STRUCT
		In : Vis_Main_In_Type;
		Internal : Vis_Main_Internal_Type;
		Out : Vis_Main_Out_Type;
	END_STRUCT;
	Vis_Process_Type : 	STRUCT
		In : Vis_Process_In_Type;
		Internal : Vis_Process_Internal_Type;
		Out : Vis_Process_Out_Type;
	END_STRUCT;
	Vis_Main_Type : 	STRUCT
		In : Vis_Main_In_Type;
		Internal : Vis_Main_Internal_Type;
		Out : Vis_Main_Out_Type;
	END_STRUCT;
END_TYPE

(*Bool Toggles for Hiding Visualiazation Elements*)

TYPE
	VisBool_Type : 	STRUCT
		P104_PV_FIT_EN : BOOL;
		P104_PV_PFIT_EN : BOOL;
		P201_PV_FIT_EN : BOOL;
		P201_PV_PFIT_EN : BOOL;
		P202_PV_FIT_EN : BOOL;
		P202_PV_PFIT_EN : BOOL;
		P203_PV_FIT_EN : BOOL;
		P203_PV_PFIT_EN : BOOL;
		P104_PV_FIT : BOOL;
		P104_PV_PFIT : BOOL;
		P201_PV_FIT : BOOL;
		P201_PV_PFIT : BOOL;
		P202_PV_FIT : BOOL;
		P202_PV_PFIT : BOOL;
		P203_PV_FIT : BOOL;
		P203_PV_PFIT : BOOL;
		P102_AUTOFLOW_ON_EN : BOOL;
		P102_AUTOFLOW_OFF_EN : BOOL;
		P103_AUTOFLOW_ON_EN : BOOL;
		P103_AUTOFLOW_OFF_EN : BOOL;
		P104_AUTOFLOW_ON_EN : BOOL;
		P104_AUTOFLOW_OFF_EN : BOOL;
		P201_AUTOFLOW_ON_EN : BOOL;
		P201_AUTOFLOW_OFF_EN : BOOL;
		P202_AUTOFLOW_ON_EN : BOOL;
		P202_AUTOFLOW_OFF_EN : BOOL;
		P203_AUTOFLOW_ON_EN : BOOL;
		P203_AUTOFLOW_OFF_EN : BOOL;
		P102_AUTOFLOW_ON : BOOL;
		P102_AUTOFLOW_OFF : BOOL;
		P103_AUTOFLOW_ON : BOOL;
		P103_AUTOFLOW_OFF : BOOL;
		P104_AUTOFLOW_ON : BOOL;
		P104_AUTOFLOW_OFF : BOOL;
		P201_AUTOFLOW_ON : BOOL;
		P201_AUTOFLOW_OFF : BOOL;
		P202_AUTOFLOW_ON : BOOL;
		P202_AUTOFLOW_OFF : BOOL;
		P203_AUTOFLOW_ON : BOOL;
		P203_AUTOFLOW_OFF : BOOL;
		P101_AUTOCAL_ON_EN : BOOL;
		P101_AUTOCAL_OFF_EN : BOOL;
		P102_AUTOCAL_ON_EN : BOOL;
		P102_AUTOCAL_OFF_EN : BOOL;
		P103_AUTOCAL_ON_EN : BOOL;
		P103_AUTOCAL_OFF_EN : BOOL;
		P104_AUTOCAL_ON_EN : BOOL;
		P104_AUTOCAL_OFF_EN : BOOL;
		P201_AUTOCAL_ON_EN : BOOL;
		P201_AUTOCAL_OFF_EN : BOOL;
		P202_AUTOCAL_ON_EN : BOOL;
		P202_AUTOCAL_OFF_EN : BOOL;
		P203_AUTOCAL_ON_EN : BOOL;
		P203_AUTOCAL_OFF_EN : BOOL;
		P101_AUTOCAL_ON : BOOL;
		P101_AUTOCAL_OFF : BOOL;
		P102_AUTOCAL_ON : BOOL;
		P102_AUTOCAL_OFF : BOOL;
		P103_AUTOCAL_ON : BOOL;
		P103_AUTOCAL_OFF : BOOL;
		P104_AUTOCAL_ON : BOOL;
		P104_AUTOCAL_OFF : BOOL;
		P201_AUTOCAL_ON : BOOL;
		P201_AUTOCAL_OFF : BOOL;
		P202_AUTOCAL_ON : BOOL;
		P202_AUTOCAL_OFF : BOOL;
		P203_AUTOCAL_ON : BOOL;
		P203_AUTOCAL_OFF : BOOL;
		P204_WARN : BOOL;
		P204_ALARM : BOOL;
		P203_WARN : BOOL;
		P203_ALARM : BOOL;
		P202_WARN : BOOL;
		P202_ALARM : BOOL;
		P201_WARN : BOOL;
		P201_ALARM : BOOL;
		P102_WARN : BOOL;
		P102_ALARM : BOOL;
		P103_WARN : BOOL;
		P103_ALARM : BOOL;
		P104_WARN : BOOL;
		P104_ALARM : BOOL;
		P102_LS : BOOL;
		P103_LS : BOOL;
		LSHH200 : BOOL;
		P204_ENABLE_OPP : BOOL;
		P203_ENABLE_OPP : BOOL;
		P202_ENABLE_OPP : BOOL;
		P201_ENABLE_OPP : BOOL;
		P201_SP : BOOL;
		P202_SP : BOOL;
		P203_SP : BOOL;
		P204_SP : BOOL;
		P201_PPM : BOOL;
		P202_PPM : BOOL;
		P203_PPM : BOOL;
		P204_PPM : BOOL;
		PMAX_MANUAL : BOOL;
		P101_DMEYELLOW : BOOL;
		P101_DMEGREEN : BOOL;
		P102_DDAGREEN : BOOL;
		P103_DDAGREEN : BOOL;
		P104_DDAGREEN : BOOL;
		P202_DDAGREEN : BOOL;
		P203_DDAGREEN : BOOL;
		P102_DDAYELLOW : BOOL;
		P103_DDAYELLOW : BOOL;
		P104_DDAYELLOW : BOOL;
		P201_DDAYELLOW : BOOL;
		P202_DDAYELLOW : BOOL;
		P203_DDAYELLOW : BOOL;
		P201_DDAGREEN : BOOL;
		P201_DDA : BOOL;
		P201_DMEYELLOW : BOOL;
		P201_DMEGREEN : BOOL;
		P201_DME : BOOL;
		P201_APPM : BOOL;
		P202_APPM : BOOL;
		P203_APPM : BOOL;
		P204_APPM : BOOL;
		FI304_MODE : BOOL;
		FI303_MODE : BOOL;
		FI302_MODE : BOOL;
		FI301_MODE : BOOL;
		FI301_MODE_OPP : BOOL;
		FI302_MODE_OPP : BOOL;
		FI303_MODE_OPP : BOOL;
		FI304_MODE_OPP : BOOL;
		XV101 : BOOL;
		XV102 : BOOL;
		XV104 : BOOL;
		XV101_ERROR : BOOL;
		XV101_OPP : BOOL;
		XV102_OPP : BOOL;
		XV103_OPP : BOOL;
		XV104_OPP : BOOL;
		XV201_OPP : BOOL;
		XV202_OPP : BOOL;
		XV203_OPP : BOOL;
		XV204_OPP : BOOL;
		P201_PTYPE_OPP : BOOL;
		P101_MODE : BOOL;
		P102_MODE : BOOL;
		P103_MODE : BOOL;
		P104_MODE : BOOL;
		P201_MODE : BOOL;
		P202_MODE : BOOL;
		P203_MODE : BOOL;
		P204_MODE : BOOL;
		HR_TYPE : BOOL;
		LR_TYPE : BOOL;
		HEARTBEAT : BOOL;
		IOSTATUS : BOOL;
		CD102_TARGETHI : REAL;
		CD102_TARGETLO : REAL;
		CD101_TARGETHI : REAL;
		CD101_TARGETLO : REAL;
		ROSTER1_DISABLE : BOOL;
		ROSTER1_ENABLE : BOOL;
		ROSTER2_DISABLE : BOOL;
		ROSTER2_ENABLE : BOOL;
		ROSTER3_DISABLE : BOOL;
		ROSTER3_ENABLE : BOOL;
		ROSTER4_DISABLE : BOOL;
		ROSTER4_ENABLE : BOOL;
		ROSTER5_DISABLE : BOOL;
		ROSTER5_ENABLE : BOOL;
		ROSTER6_DISABLE : BOOL;
		ROSTER6_ENABLE : BOOL;
		ROSTER7_DISABLE : BOOL;
		ROSTER7_ENABLE : BOOL;
		ROSTER8_DISABLE : BOOL;
		ROSTER8_ENABLE : BOOL;
		ROSTER1_DIS : BOOL;
		ROSTER1_EN : BOOL;
		ROSTER2_DIS : BOOL;
		ROSTER2_EN : BOOL;
		ROSTER3_DIS : BOOL;
		ROSTER3_EN : BOOL;
		ROSTER4_DIS : BOOL;
		ROSTER4_EN : BOOL;
		ROSTER5_DIS : BOOL;
		ROSTER5_EN : BOOL;
		ROSTER6_DIS : BOOL;
		ROSTER6_EN : BOOL;
		ROSTER7_DIS : BOOL;
		ROSTER7_EN : BOOL;
		ROSTER8_DIS : BOOL;
		ROSTER8_EN : BOOL;
		SEND_ROSTER1 : BOOL;
		SEND_ROSTER2 : BOOL;
		SEND_ROSTER3 : BOOL;
		SEND_ROSTER4 : BOOL;
		SEND_ROSTER5 : BOOL;
		SEND_ROSTER6 : BOOL;
		SEND_ROSTER7 : BOOL;
		SEND_ROSTER8 : BOOL;
	END_STRUCT;
	VisNum_Type : 	STRUCT
		P101_TOTALADJ_IN : REAL;
		P102_TOTALADJ_IN : REAL;
		P103_TOTALADJ_IN : REAL;
		P104_TOTALADJ_IN : REAL;
		P201_TOTALADJ_IN : REAL;
		P202_TOTALADJ_IN : REAL;
		P203_TOTALADJ_IN : REAL;
		P101_TOTALADJ : REAL;
		P102_TOTALADJ : REAL;
		P103_TOTALADJ : REAL;
		P104_TOTALADJ : REAL;
		P201_TOTALADJ : REAL;
		P202_TOTALADJ : REAL;
		P203_TOTALADJ : REAL;
		P101_STEPADJ_IN : REAL;
		P102_STEPADJ_IN : REAL;
		P103_STEPADJ_IN : REAL;
		P104_STEPADJ_IN : REAL;
		P201_STEPADJ_IN : REAL;
		P202_STEPADJ_IN : REAL;
		P203_STEPADJ_IN : REAL;
		P101_STEPADJ : REAL;
		P102_STEPADJ : REAL;
		P103_STEPADJ : REAL;
		P104_STEPADJ : REAL;
		P201_STEPADJ : REAL;
		P202_STEPADJ : REAL;
		P203_STEPADJ : REAL;
		P101_GAIN : REAL;
		P102_GAIN : REAL;
		P103_GAIN : REAL;
		P104_GAIN : REAL;
		P201_GAIN : REAL;
		P202_GAIN : REAL;
		P203_GAIN : REAL;
		P101_GAIN_IN : REAL;
		P102_GAIN_IN : REAL;
		P103_GAIN_IN : REAL;
		P104_GAIN_IN : REAL;
		P201_GAIN_IN : REAL;
		P202_GAIN_IN : REAL;
		P203_GAIN_IN : REAL;
	END_STRUCT;
END_TYPE

(**)

TYPE
	Recipe_type : 	STRUCT
		Contacts : RosterContact_Type;
		Notes : STRING[80];
	END_STRUCT;
	Notes_Type : 	STRUCT
		LOCATION : STRING[80];
	END_STRUCT;
END_TYPE

(**)
(*Sensors, Flowmeters, Solenoids Variables*)

TYPE
	Sensor_Variables_Type : 	STRUCT  (*Flowmeter and Other Misc Sensor Variables*)
		WASTE_LVL : BOOL; (*Waste Container Level Full Indicator*)
		SERNSORS_CONFIG : UINT; (*Datamap for sensors: DCBA >> sensor301 is type A, sensor302 is type B, sensor303 is type C, sensor304 is type D*)
		SENSOR301 : REAL; (*Sensor 301 Reading*)
		SENSOR302 : REAL; (*Sensor 302 Reading*)
		SENSOR303 : REAL; (*Sensor 303 Reading*)
		SENSOR304 : REAL; (*Sensor 304 Reading*)
		FI301 : REAL; (*Flowmeter 1 Reading*)
		FI301_QT : REAL; (*Totalized Flowmeter 1*)
		FI301_MODE : UINT; (*FI301 Mode 0 = Measure  1 = Simulation*)
		FI302 : REAL; (*Flowmeter 2 Reading*)
		FI302_QT : REAL; (*Totalized Flowmeter 2*)
		FI302_MODE : UINT; (*FI302 Mode 0 = Measure  1 = Simulation*)
		FI303 : REAL; (*Flowmeter 3 Reading*)
		FI303_QT : REAL; (*Totalized Flowmeter 3*)
		FI303_MODE : UINT; (*FI303 Mode 0 = Measure  1 = Simulation*)
		FI304 : REAL; (*Flowmeter 4 Reading*)
		FI304_QT : REAL; (*Totalized Flowmeter 4*)
		FI304_MODE : UINT; (*FI304 Mode 0 = Measure  1 = Simulation*)
		CD101 : REAL; (*Current Transducer 101*)
		CD101_SP : REAL; (*Current Transducer 101 Setpoint*)
		CD102 : REAL; (*Current Transducer 102*)
		CD102_SP : REAL; (*Current Transducer 102 Setpoint*)
		CD103 : REAL; (*Current Transducer 103*)
		CD103_SP : REAL; (*Current Transducer 103 Setpoint*)
		CD101_TI : REAL; (*Temperature After Caustic*)
		CD102_TI : REAL; (*Temperature After Hydrogen Peroxide*)
		CD103_TI : REAL; (*Temperature After Hydrogen Peroxide*)
		XV101_ENABLE : UINT; (*P101 Suction Side Solenoid Feedback Installed on Skid (0 = not installed 1 = installed)*)
		XV101 : UINT; (*P101 Suction Side Solenoid Feedback*)
		XV102 : UINT; (*P102 Off Gas Solenoid Valve*)
		XV103 : UINT; (*P103 Off Gas Solenoid Valve*)
		XV104 : UINT; (*P104 Off Gas Solenoid Valve*)
		XV201 : UINT; (*P201 Off Gas Solenoid Valve*)
		XV202 : UINT; (*P202 Off Gas Solenoid Valve*)
		XV203 : UINT; (*P203 Off Gas Solenoid Valve*)
		XV204 : UINT; (*P204 Off Gas Solenoid Valve*)
	END_STRUCT;
END_TYPE

(**)
(*Alarms*)

TYPE
	AlarmConfig_Type : 	STRUCT  (*Alarm Configuration Parameters*)
		wAC_ALARM_ENABLE_ADDR : UINT; (*Alarm Enable Status Register Address*)
		AC_ENABLE : UINT; (*Alarm and Text Enable Status*)
		AC_ALARM_ENABLE : STRING[10]; (*Alarm Enable Status*)
		wAC_TXT_ENABLE_ADDR : UINT; (*Text alerts enabled Register Address*)
		AC_TXT_ENABLE : STRING[10]; (*Text alerts enabled*)
		AC_LR_ENABLE : BOOL; (*Alarm exists on Low Rate*)
		AC_HR_ENABLE : BOOL; (*Alarm exists on High Rate*)
		AC_ACTION_ENABLE : BOOL; (*Action present and associated with alarm*)
		AC_DESCRIPTION : STRING[40]; (*Description of Alarm*)
		AC_THRESHOLD_UNIT : STRING[10]; (*Units for alarm threshold*)
		wAC_ACTION_ADDR : UINT; (*Alarm action Register Address*)
		AC_ACTION : UINT; (*Alarm action*)
		wAC_DELAY_ADDR : UINT; (*Time delay on alarming Register Address*)
		AC_DELAY : UINT; (*Time delay on alarming*)
		AC_OFFSET : UINT; (*Offset for reference to alarms list for PLC *)
		wAC_THRESHOLD_ADDR : UINT; (*Alarm threshold value Register Address*)
		AC_THRESHOLD : REAL; (*Alarm threshold value*)
	END_STRUCT;
	Alarms_Type : 	STRUCT  (*General Alarm Variables*)
		ALARM_AB1 : INT; (*General Alarm Block 1*)
		ALARM_AB2 : INT; (*General Alarm Block 2*)
		ALARM_AB3 : INT; (*General Alarm Block 3*)
		ALARM_AB4 : INT; (*General Alarm Block 4*)
		ALARM_AB5 : INT; (*General Alarm Block 5*)
		ALARM_AB6 : INT; (*General Alarm Block 6*)
		ALARM_AB7 : INT; (*General Alarm Block 7*)
		ALARM_AB8 : INT; (*General Alarm Block 8*)
		ALARM_AB9 : INT; (*General Alarm Block 9*)
		ALARM_AB10 : INT; (*General Alarm Block 10*)
		ALARM_AB11 : INT; (*General Alarm Block 11*)
		ALARM_AB12 : INT; (*General Alarm Block 12*)
		ALARM_AB13 : INT; (*General Alarm Block 13*)
		ALARM_AB14 : INT; (*General Alarm Block 14*)
		ALARM_AB15 : INT; (*General Alarm Block 15*)
		ALARM_AB16 : INT; (*General Alarm Block 16*)
		ALARM_AB17 : INT; (*General Alarm Block 17*)
		ALARM_AB18 : INT; (*General Alarm Block 18*)
		ALARM_AB19 : INT; (*General Alarm Block 19*)
	END_STRUCT;
END_TYPE

(*Status*)

TYPE
	Status_Type : 	STRUCT  (*General Alarm Variables*)
		P201_STATUS : STRING[20]; (*P201 pump status*)
		P202_STATUS : STRING[20]; (*P202 pump status*)
		P203_STATUS : STRING[20]; (*P203 pump status*)
		PMAX_HOA : STRING[20]; (*Pmax HOA  status*)
		PMAX_STATUS : STRING[20]; (*Pmax unit status*)
	END_STRUCT;
END_TYPE

(**)
(*Heartbeat*)

TYPE
	Heartbeat_Type : 	STRUCT  (*Heartbeat Connection Status Components*)
		PREVIOUS_HEARTBEAT : INT; (*Last value of heartbeat from PLC*)
		MODBUS_RESET : R_TRIG; (*Timer window to detect heartbeat*)
		UNCHANGED_TIMER : TON; (*Timer window to detect heartbeat*)
		SYSTEM_OFFLINE : BOOL; (*System Online Status (1=Offline)*)
	END_STRUCT;
END_TYPE

(**)
(*Conversion/Chem Reaction Efficiencies*)

TYPE
	ConversionRatios_Type : 	STRUCT  (*Efficiency Conversion Ratio Variables*)
		EFF_1 : REAL; (*HP to PAA Conversion Efficiency *)
		EFF_2 : REAL; (*Acetyl Conversion Efficiency *)
		TRI_TO_H2O2 : REAL; (*Molar Ratio of Triacetin to HP*)
		NAOH_TO_TRI : REAL; (*Molar Ratio of NaOH to TRI*)
		NAOH_TO_H2O2 : REAL; (*Molar Ratio of NaOH to HP*)
	END_STRUCT;
END_TYPE

(**)
(*Pmax Generation General Variables*)

TYPE
	Pmax_General_Variables_Type : 	STRUCT  (*PeroxyMax General Variables*)
		PLC_REV_A : REAL; (*PLC Revision Part A*)
		PLC_REV_B : REAL; (*PLC Revision Part B*)
		HMI_REV_A : REAL; (*HMI Revision Part A*)
		HMI_REV_B : REAL; (*HMI Revision Part B*)
		SCREEN_LOCK : BOOL; (*Unit HMI Lockout from SCADA, 1 = Locked   0 = Unlocked*)
		UNIT_ID : UINT; (*Pmax Skid ID*)
		PMAX_HOA : UINT; (*Pmax Generation is ON*)
		PMAX_STATUS : UINT; (*Pmax Status*)
		PMAX_CONC : REAL; (*Pmax Concentration*)
		PMAX_PV : REAL; (*Pmax Present Value*)
		PMAX_RATE : REAL; (*Pmax Rate*)
		HP_CONC_OD : REAL; (*HP Concentration On Deck*)
		HP_CONC : REAL; (*HP Concentration*)
		NAOH_CONC_OD : REAL; (*NaOh Concentration On Deck*)
		NAOH_CONC : REAL; (*NaOh Concentration*)
		USER_ID : UINT; (*Current Local User*)
		USER_ACCESS : UINT; (*Current Local User Access Level*)
		UNIT_TYPE : UINT; (*Unit Type ()*)
		UNIT_ID_DOSE : UINT;
		HEARTBEAT : INT; (*Unit Heartbeat*)
	END_STRUCT;
END_TYPE

(**)
(*Buffer Tank*)

TYPE
	BufferTank_Variables_Type : 	STRUCT  (*Buffer Tank Variables*)
		LSHH200 : REAL; (*Buffer Tank High High Sensor*)
		LI200P : REAL; (*Buffer Tank Level Percent*)
		LI200 : REAL; (*Buffer Tank Level*)
		DRAINTIME_SP : REAL; (*Tank Draintime Setpoint*)
		DRAINTIME_PV : REAL; (*Tank Draintime Present Value*)
		FILLTIME_SP : REAL; (*Tank Filltime Setpoint*)
		FILLTIME_PV : REAL; (*Tank Filltime Present Value*)
		BT_PERCENT : REAL; (*Buffer Tank Fill Percent*)
	END_STRUCT;
END_TYPE

(**)
(*PMAX Pumps*)

TYPE
	Pmax_Pump_101_Type : 	STRUCT  (*Pmax Generation Variables for Pump 101 - Water Pump*)
		P101_XS : UINT; (*Pump 101 On/Off Status*)
		P101_LS : REAL; (*Pump 101 Inlet Point Level*)
		P101_PFI : REAL; (*Pump 101 Feedback Percent*)
		P101_SP : REAL; (*Pump 101 Setpoint*)
		P101_PV : REAL; (*Pump 101 Current Value*)
		P101_OP : REAL; (*Pump 101 Output Percent*)
		P101_FQ : REAL; (*Pump 101 Totalized Flowmeter*)
		P101_TI : REAL; (*Pump 101 Temperature*)
		P101_PI : REAL; (*Pump 101 Pressure*)
		P101_AUTOCAL : UINT; (*Pump 101 AutoCal On/OFF Status*)
		P101_GAIN : REAL; (*Pump 101 Gain*)
		P101_STEPADJ : REAL; (*Pump 101 Max Step Adj*)
		P101_TOTALADJ : REAL; (*Pump 101 Max Total Adj*)
	END_STRUCT;
	Pmax_Pump_101B_Type : 	STRUCT  (*Pmax Generation Variables for Pump 101 - Redundant Water Pump*)
		P101B_LS : REAL; (*Pump 101B Inlet Point Level*)
		P101B_PFI : REAL; (*Pump 101B Feedback Percent*)
		P101B_SP : REAL; (*Pump 101B Setpoint*)
		P101B_OP : REAL; (*Pump 101B Output Percent*)
	END_STRUCT;
	Pmax_Pump_102_Type : 	STRUCT  (*Pmax Generation Variables for Pump 102 - Sodium Hydroxide (Caustic) Pump*)
		P102_XS : UINT; (*Pump 102 On/Off Status*)
		P102_SP : REAL; (*Pump 102 Setpoint*)
		P102_PV : REAL; (*Pump 102 Current Value*)
		P102_OP : REAL; (*Pump 102 Output Percent*)
		P102_PFI : REAL; (*Pump 102 Feedback Percent*)
		P102_FQ : REAL; (*Pump 102 Totalized Flowmeter*)
		P102_PFQ : REAL; (*Pump 102 Totalizer*)
		P102_PPI : REAL; (*Pump 102 Internal Pressure*)
		P102_TI : REAL; (*Pump 102 Temperature*)
		P102_PI : REAL; (*Pump 102 Pressure*)
		P102_ALARM : UINT; (*Pump 102 Internal Alarm Message Index*)
		P102_WARN : UINT; (*Pump 102 Internal Warning Message Index*)
		P102_LS : REAL; (*Pump 102 Inlet Point Level*)
		P102_AUTOADAPT : UINT; (*Pump 102 AutoAdapt Enable/Disable*)
		P102_AUTOCAL : UINT; (*Pump 102 AutoCal On/OFF Status*)
		P102_GAIN : REAL; (*Pump 102 Gain*)
		P102_STEPADJ : REAL; (*Pump 102 Max Step Adj*)
		P102_TOTALADJ : REAL; (*Pump 102 Max Total Adj*)
		XV102_ENABLE : UINT; (*Pump 102 XV102 Exists on Unit*)
	END_STRUCT;
	Pmax_Pump_103_Type : 	STRUCT  (*Pmax Generation Variables for Pump 103 - Hydrogen Peroxide Pump*)
		P103_XS : UINT; (*Pump 103 On/Off Status*)
		P103_SP : REAL; (*Pump 103 Setpoint*)
		P103_PV : REAL; (*Pump 103 Current Value*)
		P103_OP : REAL; (*Pump 103 Output Percent*)
		P103_PFI : REAL; (*Pump 103 Feedback Percent*)
		P103_FQ : REAL; (*Pump 103 Totalized Flowmeter*)
		P103_PFQ : REAL; (*Pump 103 Totalizer*)
		P103_PPI : REAL; (*Pump 103 Internal Pressure*)
		P103_TI : REAL; (*Pump 103 Temperature*)
		P103_PI : REAL; (*Pump 103 Pressure*)
		P103_ALARM : UINT; (*Pump 103 Internal Alarm Message Index*)
		P103_WARN : UINT; (*Pump 103 Internal Warning Message Index*)
		P103_LS : REAL; (*Pump 103 Inlet Point Level*)
		P103_AUTOADAPT : UINT; (*Pump 103 AutoAdapt Enable/Disable*)
		P103_AUTOCAL : UINT; (*Pump 103 AutoCal On/OFF Status*)
		P103_GAIN : REAL; (*Pump 103 Gain*)
		P103_STEPADJ : REAL; (*Pump 103 Max Step Adj*)
		P103_TOTALADJ : REAL; (*Pump 103 Max Total Adj*)
	END_STRUCT;
	Pmax_Pump_104_Type : 	STRUCT  (*Pmax Generation Variables for Pump 104 - Triacetin Pump*)
		P104_XS : UINT; (*Pump 104 On/Off Status*)
		P104_SP : REAL; (*Pump 104 Setpoint*)
		P104_PV : REAL; (*Pump 104 Current Value*)
		P104_OP : REAL; (*Pump 104  Output Percent*)
		P104_PFI : REAL; (*Pump 104  Feedback Percent*)
		P104_FQ : REAL; (*Pump 104 Totalized Flowmeter*)
		P104_PFQ : REAL; (*Pump 104 Totalizer*)
		P104_PI : REAL; (*Pump 104 Pressure*)
		P104_LS : REAL; (*Pump 104 Inlet Point Level*)
		P104_ALARM : UINT; (*Pump 104 Internal Alarm Message Index*)
		P104_WARN : UINT; (*Pump 104 Internal Warning Message Index*)
		P104_PPI : REAL; (*Pump 104 Internal Pressure*)
		P104_AUTOCAL : UINT; (*Pump 104 AutoCal On/OFF Status*)
		P104_AUTOADAPT : UINT; (*Pump 104 AutoAdapt Enable/Disable*)
		P104_AUTOCAL_PV : UINT; (*Pump 104 AutoCal PV Source*)
		P104_GAIN : REAL; (*Pump 104 Gain*)
		P104_STEPADJ : REAL; (*Pump 104 Max Step Adj*)
		P104_TOTALADJ : REAL; (*Pump 104 Max Total Adj*)
		XV104_ENABLE : UINT; (*Pump 104 XV104 Exists on Unit*)
	END_STRUCT;
END_TYPE

(**)
(*Dosing Pumps*)

TYPE
	Dosing_Pump_201_Type : 	STRUCT  (*Dosing Pump Variables for Dosing Pump 201*)
		P201_PTYPE : UINT; (*Pump 201 Pump Type  0 = DDA   1 = DME*)
		P201_XS : UINT; (*Pump 201 On/Off Status*)
		P201_CHEM : UINT; (*Pump 201 Chemical*)
		P201_HOA : UINT; (*Pump 201 Mode*)
		P201_PPM : REAL; (*Pump 201 Dose*)
		P201_APPM : REAL; (*Pump 201 Adjusted Dose*)
		P201_SP : REAL; (*Pump 201 Setpoint*)
		P201_PV : REAL; (*Pump 201 Present Value*)
		P201_OP : REAL; (*Pump 201 Output %*)
		P201_PFI : REAL; (*Pump 201 Feedback %*)
		P201_FQ : REAL; (*Pump 201 Totalized Flowmeter*)
		P201_PI : REAL; (*Pump 201 Pressure*)
		P201_TI : REAL; (*Pump 201 Temperature*)
		P201_PFQ : REAL; (*Pump 201 Totalizer*)
		P201_CONC : REAL; (*Pump 201 Concentration*)
		P201_REF_SENSOR : REAL; (*Pump 201 Reference Sensor*)
		P201_LS : REAL; (*Pump 201 Inlet Point Level*)
		P201_ASP : REAL; (*Pump 201 Adjusted Setpoint Value*)
		P201_PPI : REAL; (*Pump 201 Internal Pressure*)
		P201_ADJ : UINT; (*Pump 201 Adjusted Max SP Condition Present  0 = Hidden   1 = Visible*)
		P201_ALARM : UINT; (*Pump 201 Internal Alarm Message Index*)
		P201_WARN : UINT; (*Pump 201 Internal Warning Message Index*)
		P201_ENABLE : UINT; (*Pump 202 Visualization Enable Bit 0 = Visible  1 = Hidden*)
		P201_TEXT : STRING[80]; (*Pump 201 HMI Text Input Description*)
		P201_AUTOCAL : UINT; (*Pump 201 AutoCal On/OFF Status*)
		P201_AUTOADAPT : UINT; (*Pump 201 AutoAdapt Enable/Disable*)
		P201_AUTOCAL_PV : UINT; (*Pump 201 AutoCal PV Source*)
		P201_GAIN : REAL; (*Pump 201 Gain*)
		P201_STEPADJ : REAL; (*Pump 201 Max Step Adj*)
		P201_TOTALADJ : REAL; (*Pump 201 Max Total Adj*)
	END_STRUCT;
	Dosing_Pump_202_Type : 	STRUCT  (*Dosing Pump Variables for Dosing Pump 202*)
		P202_XS : UINT; (*Pump 202 On/Off Status*)
		P202_HOA : UINT; (*Pump 202 Mode*)
		P202_CHEM : UINT; (*Pump 202 Chemical*)
		P202_PPM : REAL; (*Pump 202 Dose*)
		P202_APPM : REAL; (*Pump 202 Adjusted Dose*)
		P202_SP : REAL; (*Pump 202 Setpoint*)
		P202_PV : REAL; (*Pump 202 Present Value*)
		P202_OP : REAL; (*Pump 202 Output %*)
		P202_PFI : REAL; (*Pump 202 Feedback %*)
		P202_FQ : REAL; (*Pump 202 Totalized Flowmeter*)
		P202_PI : REAL; (*Pump 202 Pressure*)
		P202_TI : REAL; (*Pump 202 Temperature*)
		P202_PFQ : REAL; (*Pump 202 Totalizer*)
		P202_CONC : REAL; (*Pump 202 Concentration*)
		P202_REF_SENSOR : REAL; (*Pump 202 Reference Sensor*)
		P202_LS : REAL; (*Pump 202 Inlet Point Level*)
		P202_PPI : REAL; (*Pump 202 Internal Pressure*)
		P202_ASP : REAL; (*Pump 202 Adjusted Setpoint Value*)
		P202_ADJ : UINT; (*Pump 202 Adjusted Max SP Condition Present  0 = Hidden   1 = Visible*)
		P202_ALARM : UINT; (*Pump 202 Internal Alarm Message Index*)
		P202_WARN : UINT; (*Pump 202 Internal Warning Message Index*)
		P202_ENABLE : UINT; (*Pump 202 Visualization Enable Bit 0 = Visible  1 = Hidden*)
		P202_TEXT : STRING[80]; (*Pump 202 HMI Text Input Description*)
		P202_AUTOCAL : UINT; (*Pump 202 AutoCal On/OFF Status*)
		P202_AUTOADAPT : UINT; (*Pump 202 AutoAdapt Enable/Disable*)
		P202_AUTOCAL_PV : UINT; (*Pump 202 AutoCal PV Source*)
		P202_GAIN : REAL; (*Pump 202 Gain*)
		P202_STEPADJ : REAL; (*Pump 202 Max Step Adj*)
		P202_TOTALADJ : REAL; (*Pump 202 Max Total Adj*)
	END_STRUCT;
	Dosing_Pump_203_Type : 	STRUCT  (*Dosing Pump Variables for Dosing Pump 203*)
		P203_XS : UINT; (*Pump 203 On/Off Status*)
		P203_HOA : UINT; (*Pump 203 Mode*)
		P203_CHEM : UINT; (*Pump 203 Chemical*)
		P203_PPM : REAL; (*Pump 203 Dose*)
		P203_APPM : REAL; (*Pump 203 Adjusted Dose*)
		P203_SP : REAL; (*Pump 203 Setpoint*)
		P203_PV : REAL; (*Pump 203 Present Value*)
		P203_OP : REAL; (*Pump 203 Output %*)
		P203_PFI : REAL; (*Pump 203 Feedback %*)
		P203_FQ : REAL; (*Pump 203 Totalized Flowmeter*)
		P203_PI : REAL; (*Pump 203 Pressure*)
		P203_TI : REAL; (*Pump 203 Temperature*)
		P203_PFQ : REAL; (*Pump 203 Totalizer*)
		P203_CONC : REAL; (*Pump 203 Concentration*)
		P203_REF_SENSOR : REAL; (*Pump 203 Reference Sensor*)
		P203_LS : REAL; (*Pump 203 Inlet Point Level*)
		P203_PPI : REAL; (*Pump 203 Internal Pressure*)
		P203_ASP : REAL; (*Pump 203 Adjusted Setpoint Value*)
		P203_ADJ : UINT; (*Pump 203 Adjusted Max SP Condition Present  0 = Hidden   1 = Visible*)
		P203_ALARM : UINT; (*Pump 203 Internal Alarm Message Index*)
		P203_WARN : UINT; (*Pump 202 Internal Warning Message Index*)
		P203_ENABLE : UINT; (*Pump 203 Visualization Enable Bit 0 = Visible  1 = Hidden*)
		P203_TEXT : STRING[80]; (*Pump 203 HMI Text Input Description*)
		P203_AUTOCAL : UINT; (*Pump 203 AutoCal On/OFF Status*)
		P203_AUTOADAPT : UINT; (*Pump 203 AutoAdapt Enable/Disable*)
		P203_AUTOCAL_PV : UINT; (*Pump 203 AutoCal PV Source*)
		P203_GAIN : REAL; (*Pump 203 Gain*)
		P203_STEPADJ : REAL; (*Pump 203 Max Step Adj*)
		P203_TOTALADJ : REAL; (*Pump 203 Max Total Adj*)
	END_STRUCT;
	Dosing_Pump_204_Type : 	STRUCT  (*Dosing Pump Variables for Dosing Pump 204*)
		P204_XS : UINT; (*Pump 204 On/Off Status*)
		P204_HOA : UINT; (*Pump 204 Mode*)
		P204_CHEM : UINT; (*Pump 204 Chemical*)
		P204_PPM : REAL; (*Pump 204 Dose*)
		P204_APPM : REAL; (*Pump 204 Adjusted Dose*)
		P204_SP : REAL; (*Pump 204 Setpoint*)
		P204_PV : REAL; (*Pump 204 Present Value*)
		P204_OP : REAL; (*Pump 204 Output %*)
		P204_PFI : REAL; (*Pump 204 Feedback %*)
		P204_FQ : REAL; (*Pump 204 Totalized Flowmeter*)
		P204_PI : REAL; (*Pump 204 Pressure*)
		P204_TI : REAL; (*Pump 204 Temperature*)
		P204_PFQ : REAL; (*Pump 204 Totalizer*)
		P204_CONC : REAL; (*Pump 204 Concentration*)
		P204_REF_SENSOR : REAL; (*Pump 204 Reference Sensor*)
		P204_LS : REAL; (*Pump 204 Inlet Point Level*)
		P204_PPI : REAL; (*Pump 204 Internal Pressure*)
		P204_ASP : REAL; (*Pump 204 Adjusted Setpoint Value*)
		P204_ADJ : UINT; (*Pump 204 Adjusted Max SP Condition Present  0 = Hidden   1 = Visible*)
		P204_ALARM : UINT; (*Pump 204 Internal Alarm Message Index*)
		P204_WARN : UINT; (*Pump 204 Internal Warning Message Index*)
		P204_ENABLE : UINT; (*Pump 204 Visualization Enable Bit 0 = Visible  1 = Hidden*)
		P204_TEXT : STRING[80]; (*Pump 204 HMI Text Input Description*)
		P204_AUTOCAL : UINT; (*Pump 204 AutoCal On/OFF Status*)
		P204_AUTOADAPT : UINT; (*Pump 204 AutoAdapt Enable/Disable*)
		P204_AUTOCAL_PV : UINT; (*Pump 204 AutoCal PV Source*)
		P204_GAIN : REAL; (*Pump 204 Gain*)
		P204_STEPADJ : REAL; (*Pump 204 Max Step Adj*)
		P204_TOTALADJ : REAL; (*Pump 204 Max Total Adj*)
	END_STRUCT;
	Dosing_Pump_205_Type : 	STRUCT  (*Dosing Pump Variables for Dosing Pump 205*)
		P205_XS : UINT; (*Pump 205 On/Off Status*)
		P205_HOA : UINT; (*Pump 205 Mode*)
		P205_CHEM : UINT; (*Pump 205 Chemical*)
		P205_PPM : REAL; (*Pump 205 Dose*)
		P205_APPM : REAL; (*Pump 205 Adjusted Dose*)
		P205_SP : REAL; (*Pump 205 Setpoint*)
		P205_PV : REAL; (*Pump 205 Present Value*)
		P205_OP : REAL; (*Pump 205 Output %*)
		P205_PFI : REAL; (*Pump 205 Feedback %*)
		P205_FQ : REAL; (*Pump 205 Totalized Flowmeter*)
		P205_PI : REAL; (*Pump 205 Pressure*)
		P205_TI : REAL; (*Pump 205 Temperature*)
		P205_PFQ : REAL; (*Pump 205 Totalizer*)
		P205_CONC : REAL; (*Pump 205 Concentration*)
		P205_REF_SENSOR : REAL; (*Pump 205 Reference Sensor*)
		P205_LS : REAL; (*Pump 205 Inlet Point Level*)
		P205_PPI : REAL; (*Pump 205 Internal Pressure*)
		P205_ASP : REAL; (*Pump 205 Adjusted Setpoint Value*)
		P205_ADJ : UINT; (*Pump 205 Adjusted Max SP Condition Present  0 = Hidden   1 = Visible*)
		P205_ALARM : UINT; (*Pump 205 Internal Alarm Message Index*)
		P205_WARN : UINT; (*Pump 205 Internal Warning Message Index*)
		P205_ENABLE : UINT; (*Pump 205 Visualization Enable Bit 0 = Visible  1 = Hidden*)
		P205_TEXT : STRING[80]; (*Pump 205 HMI Text Input Description*)
	END_STRUCT;
	Dosing_Pump_206_Type : 	STRUCT  (*Dosing Pump Variables for Dosing Pump 206*)
		P206_XS : UINT; (*Pump 206 On/Off Status*)
		P206_HOA : UINT; (*Pump 206 Mode*)
		P206_CHEM : UINT; (*Pump 206 Chemical*)
		P206_PPM : REAL; (*Pump 206 Dose*)
		P206_APPM : REAL; (*Pump 206 Adjusted Dose*)
		P206_SP : REAL; (*Pump 206 Setpoint*)
		P206_PV : REAL; (*Pump 206 Present Value*)
		P206_OP : REAL; (*Pump 206 Output %*)
		P206_PFI : REAL; (*Pump 206 Feedback %*)
		P206_FQ : REAL; (*Pump 206 Totalized Flowmeter*)
		P206_PI : REAL; (*Pump 206 Pressure*)
		P206_TI : REAL; (*Pump 206 Temperature*)
		P206_PFQ : REAL; (*Pump 206 Totalizer*)
		P206_CONC : REAL; (*Pump 206 Concentration*)
		P206_REF_SENSOR : REAL; (*Pump 206 Reference Sensor*)
		P206_LS : REAL; (*Pump 206 Inlet Point Level*)
		P206_PPI : REAL; (*Pump 206 Internal Pressure*)
		P206_ASP : REAL; (*Pump 206 Adjusted Setpoint Value*)
		P206_ADJ : UINT; (*Pump 206 Adjusted Max SP Condition Present  0 = Hidden   1 = Visible*)
		P206_ALARM : UINT; (*Pump 206 Internal Alarm Message Index*)
		P206_WARN : UINT; (*Pump 206 Internal Warning Message Index*)
		P206_ENABLE : UINT; (*Pump 206 Visualization Enable Bit 0 = Visible  1 = Hidden*)
		P206_TEXT : STRING[80]; (*Pump 206 HMI Text Input Description*)
	END_STRUCT;
	Dosing_Pump_207_Type : 	STRUCT  (*Dosing Pump Variables for Dosing Pump 207*)
		P207_XS : UINT; (*Pump 207 On/Off Status*)
		P207_HOA : UINT; (*Pump 207 Mode*)
		P207_CHEM : UINT; (*Pump 207 Chemical*)
		P207_PPM : REAL; (*Pump 207 Dose*)
		P207_APPM : REAL; (*Pump 207 Adjusted Dose*)
		P207_SP : REAL; (*Pump 207 Setpoint*)
		P207_PV : REAL; (*Pump 207 Present Value*)
		P207_OP : REAL; (*Pump 207 Output %*)
		P207_PFI : REAL; (*Pump 207 Feedback %*)
		P207_FQ : REAL; (*Pump 207 Totalized Flowmeter*)
		P207_PI : REAL; (*Pump 207 Pressure*)
		P207_TI : REAL; (*Pump 207 Temperature*)
		P207_PFQ : REAL; (*Pump 207 Totalizer*)
		P207_CONC : REAL; (*Pump 207 Concentration*)
		P207_REF_SENSOR : REAL; (*Pump 207 Reference Sensor*)
		P207_LS : REAL; (*Pump 207 Inlet Point Level*)
		P207_PPI : REAL; (*Pump 207 Internal Pressure*)
		P207_ASP : REAL; (*Pump 203 Adjusted Setpoint Value*)
		P207_ADJ : UINT; (*Pump 207 Adjusted Max SP Condition Present  0 = Hidden   1 = Visible*)
		P207_ALARM : UINT; (*Pump 207 Internal Alarm Message Index*)
		P207_WARN : UINT; (*Pump 207 Internal Warning Message Index*)
		P207_ENABLE : UINT; (*Pump 207 Visualization Enable Bit 0 = Visible  1 = Hidden*)
		P207_TEXT : STRING[80]; (*Pump 207 HMI Text Input Description*)
	END_STRUCT;
	Dosing_Pump_208_Type : 	STRUCT  (*Dosing Pump Variables for Dosing Pump 208*)
		P208_XS : UINT; (*Pump 208 On/Off Status*)
		P208_HOA : UINT; (*Pump 208 Mode*)
		P208_CHEM : UINT; (*Pump 208 Chemical*)
		P208_PPM : REAL; (*Pump 208 Dose*)
		P208_APPM : REAL; (*Pump 208 Adjusted Dose*)
		P208_SP : REAL; (*Pump 208 Setpoint*)
		P208_PV : REAL; (*Pump 208 Present Value*)
		P208_OP : REAL; (*Pump 208 Output %*)
		P208_PFI : REAL; (*Pump 208 Feedback %*)
		P208_FQ : REAL; (*Pump 208 Totalized Flowmeter*)
		P208_PI : REAL; (*Pump 208 Pressure*)
		P208_TI : REAL; (*Pump 208 Temperature*)
		P208_PFQ : REAL; (*Pump 208 Totalizer*)
		P208_CONC : REAL; (*Pump 208 Concentration*)
		P208_REF_SENSOR : REAL; (*Pump 208 Reference Sensor*)
		P208_LS : REAL; (*Pump 208 Inlet Point Level*)
		P208_PPI : REAL; (*Pump 208 Internal Pressure*)
		P208_ASP : REAL; (*Pump 208 Adjusted Setpoint Value*)
		P208_ADJ : UINT; (*Pump 208 Adjusted Max SP Condition Present  0 = Hidden   1 = Visible*)
		P208_ALARM : UINT; (*Pump 208 Internal Alarm Message Index*)
		P208_WARN : UINT; (*Pump 208 Internal Warning Message Index*)
		P208_ENABLE : UINT; (*Pump 208 Visualization Enable Bit 0 = Visible  1 = Hidden*)
		P208_TEXT : STRING[80]; (*Pump 208 HMI Text Input Description*)
	END_STRUCT;
END_TYPE

(**)
(*System Information for swapping in between different modes and functionalities*)

TYPE
	Sys_Mode_Information : 	STRUCT
		Sys_Mode : UINT; (*Mode for Visability/Changability of Variables*)
	END_STRUCT;
	ModbusDriver_Type : 	STRUCT
		BlockRecieved : BOOL;
		BlockSend : BOOL;
	END_STRUCT;
END_TYPE
```

### Services.typ - Global data types
```iecst
TYPE
	S_Recipe_type : 	STRUCT
		MpRecipeRegPar : MpRecipeRegPar;
		MpRecipeXml : MpRecipeXml;
		CreateNoteFile : BOOL;
	END_STRUCT;
	S_Alarms_global_type : 	STRUCT
		MpAlarmXListUI_0 : MpAlarmXListUI;
		MpAlarmXHistory_0 : MpAlarmXHistory;
		MpAlarmXCore_0 : MpAlarmXCore;
		MpAlarmXHistoryUI_0 : MpAlarmXHistoryUI;
		HA_AlarmXCore_0 : HA_AlarmXCore;
		AlarmList : ARRAY[0..HA_ALARMX_BUFFER_IDX]OF HA_AlarmX_Core_Buffer_typ;
	END_STRUCT;
	Services_typ : 	STRUCT
		DeviceName : STRING[255];
		Alarms_HR : ARRAY[0..MAX_SKIDS_HR]OF S_Alarms_typ;
		Alarms_LR : ARRAY[0..MAX_SKIDS_LR]OF S_Alarms_typ;
		Alarms_Global : S_Alarms_global_type;
		Recipe : S_Recipe_type;
	END_STRUCT;
	S_Alarms_typ : 	STRUCT
		In : S_Alarms_In_typ;
		Internal : S_Alarms_Internal_typ;
		Out : S_Alarms_Out_typ;
	END_STRUCT;
	S_Alarms_In_typ : 	STRUCT
		ResetAlarms : BOOL;
		ClearHistory : BOOL;
		ExportHistory : BOOL;
		AlarmList : ARRAY[0..HA_ALARMX_BUFFER_IDX]OF HA_AlarmX_Core_Buffer_typ;
	END_STRUCT;
	S_Alarms_Internal_typ : 	STRUCT
		MpAlarmXListUI_0 : MpAlarmXListUI;
		MpAlarmXHistory_0 : MpAlarmXHistory;
		MpAlarmXCore_0 : MpAlarmXCore;
		CTON_ResetDelay : CTON;
		StateResetAlarms : INT;
		StateExportHistory : INT;
		MpAlarmXHistoryUI_0 : MpAlarmXHistoryUI;
		HA_AlarmXCore_0 : HA_AlarmXCore;
		Alarms_State : Alarms_Type;
		Alarm_Set_Delay : TON;
	END_STRUCT;
	S_Alarms_Out_typ : 	STRUCT
		AlarmActive : BOOL;
		BufferInfo : HA_AlarmX_BufferInfo_typ;
	END_STRUCT;
END_TYPE
```

### Package Logical/Libraries - Global libraries

### Library Logical/Libraries/Str2DtPvdr (IEC)

#### Str2DtPvdr.fun
```iecst
{REDUND_ERROR} FUNCTION WString2DataProvider : BOOL (*TODO: Add your comment here*) (*$GROUP=User,$CAT=User,$GROUPICON=User.png,$CATICON=User.png*)
	VAR_INPUT
		SourceString : UDINT;
		Value : UDINT;
		TargetString : UDINT;
	END_VAR
	VAR
		Value_String : WSTRING[40];
	END_VAR
END_FUNCTION

FUNCTION StepListElementCreator : BOOL
	VAR_INPUT
		SourceString : UDINT;
		Index : DINT;
		TargetString : UDINT;
	END_VAR
	VAR
		IndexString : STRING[80];
		IndexWString : WSTRING[80];
	END_VAR
END_FUNCTION

{REDUND_ERROR} FUNCTION String2DataProvider : BOOL (*TODO: Add your comment here*) (*$GROUP=User,$CAT=User,$GROUPICON=User.png,$CATICON=User.png*)
	VAR_INPUT
		SourceString : UDINT;
		TargetString : UDINT;
	END_VAR
END_FUNCTION
```

#### Str2DtPvdr.st
```iecst
(* TODO: Add your comment here *)
FUNCTION WString2DataProvider

	brwcscpy(TargetString, ADR("{$"value$":$""));
	Value_String := UDINT_TO_WSTRING(Value);
	brwcscat(TargetString, ADR(Value_String));
	brwcscat(TargetString, ADR("$",$"text$":$""));
	brwcscat(TargetString, SourceString);
	brwcscat(TargetString, ADR("$"}"));

	WString2DataProvider := TRUE;
END_FUNCTION

FUNCTION String2DataProvider
	brsstrcpy (TargetString, ADR('{$'value$':$''));
	brsstrcat(TargetString, SourceString);
	brsstrcat(TargetString, ADR('$',$'text$':$''));
	brsstrcat(TargetString, SourceString);
	brsstrcat(TargetString, ADR('$'}'));

	String2DataProvider := TRUE;
END_FUNCTION

FUNCTION StepListElementCreator
	brwcscpy(TargetString, ADR("Step "));
	brsitoa(Index,ADR(IndexString));
	IndexWString:=STRING_TO_WSTRING(IndexString);
	brwcscat(TargetString, ADR(IndexWString));
	brwcscat(TargetString, ADR(": "));
	brwcscat(TargetString, SourceString);

	StepListElementCreator := TRUE;
END_FUNCTION
```

- Project.language (not shown)

### Library Logical/Libraries/HA_IO (IEC)

#### Types.typ - Exported data types
```iecst
TYPE
	HA_IO_Digital_Sim_typ : 	STRUCT
		Active : BOOL;
		Logical : BOOL;
	END_STRUCT;
	HA_IO_Digital_Signal_typ : 	STRUCT
		Logical : BOOL;
		EdgePosLogical : BOOL;
		EdgeNegLogical : BOOL;
		Filtered : BOOL;
		EdgePosFiltered : BOOL;
		EdgeNegFiltered : BOOL;
		IOMapping : BOOL;
		InvertedIOMapping : BOOL;
		VisIOMapping : BOOL;
		VisRefresher : BOOL;
	END_STRUCT;
	HA_IO_Digital_Par_LimitSet_typ : 	STRUCT
		FilterOnTime_Min : LREAL;
		FilterOnTime_Max : LREAL;
		FilterOffTime_Min : LREAL;
		FilterOffTime_Max : LREAL;
	END_STRUCT;
	HA_IO_Digital_Par_typ : 	STRUCT
		InvertedIOMapping : BOOL;
		FilterOnTime : LREAL;
		FilterOffTime : LREAL;
	END_STRUCT;
	HA_IO_Digital_Internal_typ : 	STRUCT
		StatusLogical : BOOL;
		StatusFiltered : BOOL;
		CTON_DB_Off : CTON;
		CTON_DB_On : CTON;
	END_STRUCT;
	HA_IO_Digital_Forcing_typ : 	STRUCT
		Off : BOOL;
		On : BOOL;
	END_STRUCT;
	HA_IO_Analog_Sim_typ : 	STRUCT
		Active : BOOL;
		Logical : LREAL;
	END_STRUCT;
	HA_IO_Analog_Signal_typ : 	STRUCT
		UnlimitedLogical : LREAL;
		MinExceeded : BOOL;
		MaxExceeded : BOOL;
		Logical : LREAL;
		Filtered : LREAL;
		Vis : HA_IO_Analog_Vis_typ;
		IOMapping : HA_IO_Analog_Mapping_typ;
	END_STRUCT;
	HA_IO_Analog_Par_LimitSet_typ : 	STRUCT
		M_Min : LREAL;
		M_Max : LREAL;
		B_Min : LREAL;
		B_Max : LREAL;
		Filter_Min : LREAL;
		Filter_Max : LREAL;
		MinValue_Min : LREAL;
		MinValue_Max : LREAL;
		MaxValue_Min : LREAL;
		MaxValue_Max : LREAL;
	END_STRUCT;
	HA_IO_Analog_Par_typ : 	STRUCT
		M : LREAL;
		B : LREAL;
		Filter : LREAL;
		MaxValue : LREAL;
		MinValue : LREAL;
	END_STRUCT;
	HA_IO_Analog_Internal_typ : 	STRUCT
		InitFilter : BOOL;
		Filter : LREAL;
		LastFilter : LREAL;
		Temp : LREAL;
	END_STRUCT;
	HA_IO_Analog_Forcing_typ : 	STRUCT
		Off : BOOL;
		On : BOOL;
		Value : LREAL;
	END_STRUCT;
	HA_IO_Analog_Vis_typ : 	STRUCT
		Raw : LREAL;
		IO : LREAL;
		App : LREAL;
	END_STRUCT;
	HA_IO_Analog_Mapping_typ : 	STRUCT
		VarSINT : SINT;
		VarUSINT : USINT;
		VarINT : INT;
		VarUINT : UINT;
		VarDINT : DINT;
		VarUDINT : UDINT;
		VarREAL : REAL;
		VarLREAL : LREAL;
	END_STRUCT;
	HA_IO_ANALOG_TYPE_ENUM :
		(
		HA_IO_ANALOG_TYPE_INT,
		HA_IO_ANALOG_TYPE_USINT,
		HA_IO_ANALOG_TYPE_SINT,
		HA_IO_ANALOG_TYPE_UINT,
		HA_IO_ANALOG_TYPE_DINT,
		HA_IO_ANALOG_TYPE_UDINT,
		HA_IO_ANALOG_TYPE_REAL,
		HA_IO_ANALOG_TYPE_LREAL
		);
END_TYPE
```

#### HA_IO.fun - Exported functions and function blocks
```iecst
{REDUND_ERROR} FUNCTION_BLOCK HA_IO_DO (* *) (*$GROUP=User,$CAT=User,$GROUPICON=User.png,$CATICON=User.png*)
	VAR_INPUT
		Logical : BOOL;
		Forcing : HA_IO_Digital_Forcing_typ;
		Par : HA_IO_Digital_Par_typ;
	END_VAR
	VAR_OUTPUT
		Signal : HA_IO_Digital_Signal_typ;
	END_VAR
	VAR
		Internal : HA_IO_Digital_Internal_typ;
	END_VAR
END_FUNCTION_BLOCK

{REDUND_ERROR} FUNCTION_BLOCK HA_IO_DI (* *) (*$GROUP=User,$CAT=User,$GROUPICON=User.png,$CATICON=User.png*)
	VAR_INPUT
		IOMapping : BOOL;
		Forcing : HA_IO_Digital_Forcing_typ;
		Par : HA_IO_Digital_Par_typ;
		Sim : HA_IO_Digital_Sim_typ;
	END_VAR
	VAR_OUTPUT
		Signal : HA_IO_Digital_Signal_typ;
	END_VAR
	VAR
		Internal : HA_IO_Digital_Internal_typ;
	END_VAR
END_FUNCTION_BLOCK

{REDUND_ERROR} FUNCTION_BLOCK HA_IO_AI (* *) (*$GROUP=User,$CAT=User,$GROUPICON=User.png,$CATICON=User.png*)
	VAR_INPUT
		VarType : HA_IO_ANALOG_TYPE_ENUM;
		IOMapping : HA_IO_Analog_Mapping_typ;
		Forcing : HA_IO_Analog_Forcing_typ;
		Sim : HA_IO_Analog_Sim_typ;
		Par : HA_IO_Analog_Par_typ;
	END_VAR
	VAR_OUTPUT
		Signal : HA_IO_Analog_Signal_typ;
	END_VAR
	VAR
		Internal : HA_IO_Analog_Internal_typ;
	END_VAR
END_FUNCTION_BLOCK

{REDUND_ERROR} FUNCTION_BLOCK HA_IO_AO (* *) (*$GROUP=User,$CAT=User,$GROUPICON=User.png,$CATICON=User.png*)
	VAR_INPUT
		VarType : HA_IO_ANALOG_TYPE_ENUM;
		Logical : LREAL;
		Forcing : HA_IO_Analog_Forcing_typ;
		Par : HA_IO_Analog_Par_typ;
	END_VAR
	VAR_OUTPUT
		Signal : HA_IO_Analog_Signal_typ;
	END_VAR
	VAR
		Internal : HA_IO_Analog_Internal_typ;
	END_VAR
END_FUNCTION_BLOCK
```

#### HA_IO_DI.st
```iecst
(* Full Digital Input Handler*)
FUNCTION_BLOCK HA_IO_DI

//LOGICAL/INVERT
	Signal.IOMapping					:= IOMapping;
	Signal.InvertedIOMapping			:= NOT Signal.IOMapping;
	IF Par.InvertedIOMapping THEN
		Signal.Logical					:= Signal.InvertedIOMapping;
	ELSE
		Signal.Logical					:= Signal.IOMapping;
	END_IF;
//SIMULATION
	IF Sim.Active THEN
		Signal.Logical					:= Sim.Logical;
		Signal.IOMapping				:= Sim.Logical;
		Signal.InvertedIOMapping		:= NOT Sim.Logical;
	END_IF;
//VISUALIZATION
	IF Par.InvertedIOMapping THEN
		Signal.VisIOMapping				:= Signal.InvertedIOMapping;
	ELSE
		Signal.VisIOMapping				:= Signal.IOMapping;
	END_IF;
//DEBOUNCING
	IF Signal.Logical THEN
		Internal.CTON_DB_Off(IN := FALSE);
		IF Internal.CTON_DB_On.Q OR Par.FilterOnTime <= 0.0 THEN
			Signal.Filtered			:= TRUE;
		ELSE
			Internal.CTON_DB_On(IN := TRUE, PT := LREAL_TO_TIME(Par.FilterOnTime*1000.0));
		END_IF;
	ELSE
		Internal.CTON_DB_On(IN := FALSE);
		IF Internal.CTON_DB_Off.Q OR Par.FilterOffTime <= 0.0 THEN
			Signal.Filtered			:= FALSE;
		ELSE
			Internal.CTON_DB_Off(IN := TRUE, PT := LREAL_TO_TIME(Par.FilterOffTime*1000.0));
		END_IF;
	END_IF;
//FORCING
	IF Forcing.On XOR Forcing.Off THEN
		IF Forcing.Off THEN
			Signal.Logical				:= FALSE;
			Signal.Filtered			:= FALSE;
		ELSIF Forcing.On THEN
			Signal.Logical				:= TRUE;
			Signal.Filtered			:= TRUE;
		END_IF;
	END_IF;
//EDGES
	Signal.EdgeNegLogical				:= FALSE;
	IF Internal.StatusLogical AND NOT Signal.Logical THEN
		Signal.EdgeNegLogical			:= TRUE;
	END_IF;
	Signal.EdgePosLogical				:= FALSE;
	IF NOT Internal.StatusLogical AND Signal.Logical THEN
		Signal.EdgePosLogical			:= TRUE;
	END_IF;
	Internal.StatusLogical 				:= Signal.Logical;

	Signal.EdgeNegFiltered				:= FALSE;
	IF Internal.StatusFiltered AND NOT Signal.Filtered THEN
		Signal.EdgeNegFiltered			:= TRUE;
	END_IF;
	Signal.EdgePosFiltered				:= FALSE;
	IF NOT Internal.StatusFiltered AND Signal.Filtered THEN
		Signal.EdgePosFiltered			:= TRUE;
	END_IF;
	Internal.StatusFiltered 			:= Signal.Filtered;

//This is needed as a workaround for an event bug that wouldnt show IO status colors if IO was active at start of Vis
	Signal.VisRefresher					:= FALSE;

END_FUNCTION_BLOCK
```

#### HA_IO_DO.st
```iecst
(* Full Digital Output Handler*)
FUNCTION_BLOCK HA_IO_DO

//LOGICAL
	Signal.Logical						:= Logical;
//DEBOUNCING
	IF Signal.Logical THEN
		Internal.CTON_DB_Off(IN := FALSE);
		IF Internal.CTON_DB_On.Q OR Par.FilterOnTime <= 0.0 THEN
			Signal.Filtered			:= TRUE;
		ELSE
			Internal.CTON_DB_On(IN := TRUE, PT := LREAL_TO_TIME(Par.FilterOnTime*1000.0));
		END_IF;
	ELSE
		Internal.CTON_DB_On(IN := FALSE);
		IF Internal.CTON_DB_Off.Q OR Par.FilterOffTime <= 0.0 THEN
			Signal.Filtered			:= FALSE;
		ELSE
			Internal.CTON_DB_Off(IN := TRUE, PT := LREAL_TO_TIME(Par.FilterOffTime*1000.0));
		END_IF;
	END_IF;
//EDGES
	Signal.EdgeNegLogical				:= FALSE;
	IF Internal.StatusLogical AND NOT Signal.Logical THEN
		Signal.EdgeNegLogical			:= TRUE;
	END_IF;
	Signal.EdgePosLogical				:= FALSE;
	IF NOT Internal.StatusLogical AND Signal.Logical THEN
		Signal.EdgePosLogical			:= TRUE;
	END_IF;
	Internal.StatusLogical 				:= Signal.Logical;

	Signal.EdgeNegFiltered				:= FALSE;
	IF Internal.StatusFiltered AND NOT Signal.Filtered THEN
		Signal.EdgeNegFiltered			:= TRUE;
	END_IF;
	Signal.EdgePosFiltered				:= FALSE;
	IF NOT Internal.StatusFiltered AND Signal.Filtered THEN
		Signal.EdgePosFiltered			:= TRUE;
	END_IF;
	Internal.StatusFiltered 			:= Signal.Filtered;
//FORCING
	Signal.IOMapping					:= Signal.Filtered;
	IF Forcing.On XOR Forcing.Off THEN
		IF Forcing.Off THEN
			Signal.IOMapping			:= FALSE;
		ELSIF Forcing.On THEN
			Signal.IOMapping			:= TRUE;
		END_IF;
	END_IF;
//INVERT
	Signal.InvertedIOMapping			:= NOT Signal.IOMapping;
//VISUALIZATION
	IF Par.InvertedIOMapping THEN
		Signal.VisIOMapping				:= Signal.InvertedIOMapping;
	ELSE
		Signal.VisIOMapping				:= Signal.IOMapping;
	END_IF;

//This is needed as a workaround for an event bug that wouldnt show IO status colors if IO was active at start of Vis
	Signal.VisRefresher					:= FALSE;

END_FUNCTION_BLOCK
```

#### HA_IO_AO.st
```iecst
(* Full Analog Output Handler*)
FUNCTION_BLOCK HA_IO_AO
//LOGICAL
	Signal.Logical						:= Logical;
	Signal.UnlimitedLogical				:= Logical;
	Signal.Vis.App						:= Logical;
	Internal.Temp						:= Logical;
//FORCING
	IF Forcing.On XOR Forcing.Off THEN
		IF Forcing.Off THEN
			Internal.Temp				:= 0.0;
		ELSIF Forcing.On THEN
			Internal.Temp				:= Forcing.Value;
		END_IF;
	END_IF;
//LIMITING
	Signal.MaxExceeded					:= FALSE;
	IF Internal.Temp > Par.MaxValue THEN
		Signal.MaxExceeded				:= TRUE;
		Internal.Temp					:= Par.MaxValue;
	END_IF;
	Signal.MinExceeded					:= FALSE;
	IF Signal.Logical < Par.MinValue THEN
		Signal.MinExceeded				:= TRUE;
		Internal.Temp					:= Par.MinValue;
	END_IF;
//FILTERING
	Internal.Filter 					:= Par.Filter;
	IF Par.Filter < 0.0 THEN
		Internal.Filter 				:= 0.0;
	ELSIF Internal.Filter > 1.0 THEN
		Internal.Filter 				:= 0.99999999;
	END_IF;
	IF NOT Internal.InitFilter OR Internal.LastFilter <> Internal.Filter THEN
		Internal.InitFilter				:= TRUE;
		Internal.LastFilter 			:= Internal.Filter;
		Signal.Filtered 				:= Internal.Temp;
	ELSE
		Signal.Filtered 				:= Internal.Temp*(1.0-Internal.Filter) + Signal.Filtered*Internal.Filter;
	END_IF;
	IF Signal.Filtered > Par.MaxValue THEN
		Signal.Filtered 				:= Par.MaxValue;
	ELSIF Signal.Filtered < Par.MinValue THEN
		Signal.Filtered 				:= Par.MinValue;
	END_IF;
//IOMAPPING
	Signal.Vis.IO						:= Signal.Filtered;
	IF Par.M <> 0 THEN
		Signal.Vis.Raw		 			:= (Signal.Filtered-Par.B)/Par.M;
	ELSE
		Signal.Vis.Raw 					:= 0.0;
	END_IF;
	CASE VarType OF
		HA_IO_ANALOG_TYPE_INT:
			Signal.IOMapping.VarINT		:= LREAL_TO_INT(Signal.Vis.Raw);
		HA_IO_ANALOG_TYPE_USINT:
			Signal.IOMapping.VarUSINT	:= LREAL_TO_USINT(Signal.Vis.Raw);
		HA_IO_ANALOG_TYPE_SINT:
			Signal.IOMapping.VarSINT	:= LREAL_TO_SINT(Signal.Vis.Raw);
		HA_IO_ANALOG_TYPE_UINT:
			Signal.IOMapping.VarUINT	:= LREAL_TO_UINT(Signal.Vis.Raw);
		HA_IO_ANALOG_TYPE_DINT:
			Signal.IOMapping.VarDINT	:= LREAL_TO_DINT(Signal.Vis.Raw);
		HA_IO_ANALOG_TYPE_UDINT:
			Signal.IOMapping.VarUDINT	:= LREAL_TO_UDINT(Signal.Vis.Raw);
		HA_IO_ANALOG_TYPE_REAL:
			Signal.IOMapping.VarREAL	:= LREAL_TO_REAL(Signal.Vis.Raw);
		HA_IO_ANALOG_TYPE_LREAL:
			Signal.IOMapping.VarLREAL	:= Signal.Vis.Raw;
	END_CASE

END_FUNCTION_BLOCK
```

#### HA_IO_AI.st
```iecst
(* Full Analog Input Handler*)
FUNCTION_BLOCK HA_IO_AI

	CASE VarType OF
		HA_IO_ANALOG_TYPE_INT:
		//LOGICAL
			Signal.IOMapping.VarINT					:= IOMapping.VarINT;
			Signal.Vis.Raw							:= INT_TO_LREAL(Signal.IOMapping.VarINT);
			Signal.Vis.IO							:= Par.M*INT_TO_LREAL(Signal.IOMapping.VarINT)+Par.B;
		//SIMULATION
			IF Sim.Active THEN
				Signal.Vis.IO						:= Sim.Logical;
				IF Par.M <> 0 THEN
					Signal.Vis.Raw					:= (Signal.Vis.IO-Par.B)/Par.M;
					Signal.IOMapping.VarINT			:= LREAL_TO_INT(Signal.Vis.Raw);
				ELSE
					Signal.Vis.Raw					:= 0.0;
					Signal.IOMapping.VarINT			:= 0;
				END_IF;
			END_IF;
		HA_IO_ANALOG_TYPE_USINT:
		//LOGICAL
			Signal.IOMapping.VarUSINT				:= IOMapping.VarUSINT;
			Signal.Vis.Raw							:= USINT_TO_LREAL(Signal.IOMapping.VarUSINT);
			Signal.Vis.IO							:= Par.M*USINT_TO_LREAL(Signal.IOMapping.VarUSINT)+Par.B;
		//SIMULATION
			IF Sim.Active THEN
				Signal.Vis.IO						:= Sim.Logical;
				IF Par.M <> 0 THEN
					Signal.Vis.Raw					:= (Signal.Vis.IO-Par.B)/Par.M;
					Signal.IOMapping.VarUSINT		:= LREAL_TO_USINT(Signal.Vis.Raw);
				ELSE
					Signal.Vis.Raw					:= 0.0;
					Signal.IOMapping.VarUSINT		:= 0;
				END_IF;
			END_IF;
		HA_IO_ANALOG_TYPE_SINT:
		//LOGICAL
			Signal.IOMapping.VarSINT				:= IOMapping.VarSINT;
			Signal.Vis.Raw							:= SINT_TO_LREAL(Signal.IOMapping.VarSINT);
			Signal.Vis.IO							:= Par.M*SINT_TO_LREAL(Signal.IOMapping.VarSINT)+Par.B;
		//SIMULATION
			IF Sim.Active THEN
				Signal.Vis.IO						:= Sim.Logical;
				IF Par.M <> 0 THEN
					Signal.Vis.Raw					:= (Signal.Vis.IO-Par.B)/Par.M;
					Signal.IOMapping.VarSINT		:= LREAL_TO_SINT(Signal.Vis.Raw);
				ELSE
					Signal.Vis.Raw					:= 0.0;
					Signal.IOMapping.VarSINT		:= 0;
				END_IF;
			END_IF;
		HA_IO_ANALOG_TYPE_UINT:
		//LOGICAL
			Signal.IOMapping.VarUINT				:= IOMapping.VarUINT;
			Signal.Vis.Raw							:= UINT_TO_LREAL(Signal.IOMapping.VarUINT);
			Signal.Vis.IO							:= Par.M*UINT_TO_LREAL(Signal.IOMapping.VarUINT)+Par.B;
		//SIMULATION
			IF Sim.Active THEN
				Signal.Vis.IO						:= Sim.Logical;
				IF Par.M <> 0 THEN
					Signal.Vis.Raw					:= (Signal.Vis.IO-Par.B)/Par.M;
					Signal.IOMapping.VarUINT		:= LREAL_TO_UINT(Signal.Vis.Raw);
				ELSE
					Signal.Vis.Raw					:= 0.0;
					Signal.IOMapping.VarUINT		:= 0;
				END_IF;
			END_IF;
		HA_IO_ANALOG_TYPE_DINT:
		//LOGICAL
			Signal.IOMapping.VarDINT				:= IOMapping.VarDINT;
			Signal.Vis.Raw							:= DINT_TO_LREAL(Signal.IOMapping.VarDINT);
			Signal.Vis.IO							:= Par.M*DINT_TO_LREAL(Signal.IOMapping.VarDINT)+Par.B;
		//SIMULATION
			IF Sim.Active THEN
				Signal.Vis.IO						:= Sim.Logical;
				IF Par.M <> 0 THEN
					Signal.Vis.Raw					:= (Signal.Vis.IO-Par.B)/Par.M;
					Signal.IOMapping.VarDINT		:= LREAL_TO_DINT(Signal.Vis.Raw);
				ELSE
					Signal.Vis.Raw					:= 0.0;
					Signal.IOMapping.VarDINT		:= 0;
				END_IF;
			END_IF;
		HA_IO_ANALOG_TYPE_UDINT:
		//LOGICAL
			Signal.IOMapping.VarUDINT				:= IOMapping.VarUDINT;
			Signal.Vis.Raw							:= UDINT_TO_LREAL(Signal.IOMapping.VarUDINT);
			Signal.Vis.IO							:= Par.M*UDINT_TO_LREAL(Signal.IOMapping.VarUDINT)+Par.B;
		//SIMULATION
			IF Sim.Active THEN
				Signal.Vis.IO						:= Sim.Logical;
				IF Par.M <> 0 THEN
					Signal.Vis.Raw					:= (Signal.Vis.IO-Par.B)/Par.M;
					Signal.IOMapping.VarUDINT		:= LREAL_TO_UDINT(Signal.Vis.Raw);
				ELSE
					Signal.Vis.Raw					:= 0.0;
					Signal.IOMapping.VarUDINT		:= 0;
				END_IF;
			END_IF;
		HA_IO_ANALOG_TYPE_REAL:
		//LOGICAL
			Signal.IOMapping.VarREAL				:= IOMapping.VarREAL;
			Signal.Vis.Raw							:= REAL_TO_LREAL(Signal.IOMapping.VarREAL);
			Signal.Vis.IO							:= Par.M*REAL_TO_LREAL(Signal.IOMapping.VarREAL)+Par.B;
		//SIMULATION
			IF Sim.Active THEN
				Signal.Vis.IO						:= Sim.Logical;
				IF Par.M <> 0 THEN
					Signal.Vis.Raw					:= (Signal.Vis.IO-Par.B)/Par.M;
					Signal.IOMapping.VarREAL		:= LREAL_TO_REAL(Signal.Vis.Raw);
				ELSE
					Signal.Vis.Raw					:= 0.0;
					Signal.IOMapping.VarREAL		:= 0;
				END_IF;
			END_IF;
		HA_IO_ANALOG_TYPE_LREAL:
		//LOGICAL
			Signal.IOMapping.VarLREAL				:= IOMapping.VarLREAL;
			Signal.Vis.Raw							:= Signal.IOMapping.VarLREAL;
			Signal.Vis.IO							:= Par.M*Signal.IOMapping.VarLREAL+Par.B;
		//SIMULATION
			IF Sim.Active THEN
				Signal.Vis.IO						:= Sim.Logical;
				IF Par.M <> 0 THEN
					Signal.Vis.Raw					:= (Signal.Vis.IO-Par.B)/Par.M;
					Signal.IOMapping.VarLREAL		:= Signal.Vis.Raw;
				ELSE
					Signal.Vis.Raw					:= 0.0;
					Signal.IOMapping.VarLREAL		:= 0;
				END_IF;
			END_IF;
	END_CASE;
	Signal.Logical									:= Signal.Vis.IO;
//FORCING
	IF Forcing.On XOR Forcing.Off THEN
		IF Forcing.Off THEN
			Signal.Logical							:= 0.0;
		ELSIF Forcing.On THEN
			Signal.Logical							:= Forcing.Value;
		END_IF;
	END_IF;
//LIMITING
	Signal.UnlimitedLogical							:= Signal.Logical;
	Signal.MaxExceeded								:= FALSE;
	IF Signal.Logical > Par.MaxValue THEN
		Signal.MaxExceeded							:= TRUE;
		Signal.Logical								:= Par.MaxValue;
	END_IF;
	Signal.MinExceeded								:= FALSE;
	IF Signal.Logical < Par.MinValue THEN
		Signal.MinExceeded							:= TRUE;
		Signal.Logical								:= Par.MinValue;
	END_IF;
//FILTERING
	Internal.Filter 								:= Par.Filter;
	IF Par.Filter < 0.0 THEN
		Internal.Filter 							:= 0.0;
	ELSIF Internal.Filter > 1.0 THEN
		Internal.Filter 							:= 0.99999999;
	END_IF;
	IF NOT Internal.InitFilter OR Internal.LastFilter <> Internal.Filter THEN
		Internal.InitFilter							:= TRUE;
		Internal.LastFilter 						:= Internal.Filter;
		Signal.Filtered 							:= Signal.Logical;
	ELSE
		Signal.Filtered 							:= Signal.Logical*(1.0-Internal.Filter) + Signal.Filtered*Internal.Filter;
	END_IF;
	IF Signal.Filtered > Par.MaxValue THEN
		Signal.Filtered 							:= Par.MaxValue;
	ELSIF Signal.Filtered < Par.MinValue THEN
		Signal.Filtered 							:= Par.MinValue;
	END_IF;
	Signal.Vis.App									:= Signal.Filtered;
END_FUNCTION_BLOCK
```

### Library Logical/Libraries/HA (IEC)

#### Types.typ - Exported data types
```iecst
TYPE
	HA_TypeSelect_typ : 	STRUCT
		Select : HA_TYPE_ENUM;
		VarSINT : SINT;
		VarUSINT : USINT;
		VarINT : INT;
		VarUINT : UINT;
		VarDINT : DINT;
		VarUDINT : UDINT;
		VarREAL : REAL;
		VarLREAL : LREAL;
		VarTIME : TIME;
		VarDT : DATE_AND_TIME;
		VarSTRING_ADR : UDINT;
		VarSTRING_LEN : UDINT;
		VarWSTRING_ADR : UDINT;
		VarWSTRING_LEN : UDINT;
	END_STRUCT;
	HA_TYPE_ENUM :
		(
		HA_TYPE_INT,
		HA_TYPE_USINT,
		HA_TYPE_SINT,
		HA_TYPE_UINT,
		HA_TYPE_DINT,
		HA_TYPE_UDINT,
		HA_TYPE_REAL,
		HA_TYPE_LREAL,
		HA_TYPE_TIME,
		HA_TYPE_DT,
		HA_TYPE_STRING,
		HA_TYPE_WSTRING
		);
END_TYPE
```

#### HA.fun - Exported functions and function blocks
```iecst
FUNCTION_BLOCK CTON
	VAR_INPUT
		IN : BOOL;
		PT : TIME;
		PAUSE : BOOL;
	END_VAR
	VAR_OUTPUT
		ET : TIME;
		Q : BOOL;
	END_VAR
	VAR
		RTInfo_0 : RTInfo;
		delta : LREAL;
		counter : LREAL;
	END_VAR
END_FUNCTION_BLOCK
```

#### CTON.st
```iecst
(* Mimic a TON block with a counter instead of a timestamp basis *)
FUNCTION_BLOCK CTON

	IF delta < 1 THEN
		RTInfo_0(enable := TRUE);
		delta := UDINT_TO_LREAL(RTInfo_0.cycle_time);
	END_IF;
	IF IN THEN
		IF (TIME_TO_LREAL(PT)*1000.0) <= (counter*delta) THEN
			Q := TRUE;
		ELSE
			IF NOT PAUSE THEN
				counter := counter + 1.0;
			END_IF;
		END_IF;
		ET := LREAL_TO_TIME((counter*delta)/1000.0);
	ELSE
		counter := 0.0;
		Q := FALSE;
		ET := 0;
	END_IF;

END_FUNCTION_BLOCK
```

### Library Logical/Libraries/HA_Version (IEC, version 1.00.0)
Depends on: ArEventLog, ArProject, AsBrStr

#### Types.typ - Exported data types
```iecst
TYPE
	IdentifyConfig_Internal_typ : 	STRUCT
		state : INT;
		AddData : STRING[500];
		ArProjectGetInfo_0 : ArProjectGetInfo;
		ArEventLogWrite_0 : ArEventLogWrite;
		ArEventLogGetIdent_0 : ArEventLogGetIdent;
	END_STRUCT;
END_TYPE
```

#### HA_Version.fun - Exported functions and function blocks
```iecst
{REDUND_ERROR} FUNCTION_BLOCK IdentifyConfig (*returns the ID and Version of the configuration as strings and also enters a record in the log book*) (*$GROUP=User,$CAT=User,$GROUPICON=User.png,$CATICON=User.png*)
	VAR_OUTPUT
		Done : BOOL;
		ConfigID : STRING[255];
		ConfigVersion : STRING[32];
	END_VAR
	VAR
		internal : IdentifyConfig_Internal_typ;
	END_VAR
END_FUNCTION_BLOCK
```

#### IdentifyConfig.st
```iecst
(* returns the ID and Version of the configuration as strings and also enters a record in the log book *)
FUNCTION_BLOCK IdentifyConfig
	Done := FALSE;
	CASE internal.state OF
		0:
			IF internal.ArProjectGetInfo_0.Done THEN
				ConfigID := internal.ArProjectGetInfo_0.ConfigurationID;
				ConfigVersion := internal.ArProjectGetInfo_0.ConfigurationVersion;
				internal.AddData := '';
				brsstrcat(ADR(internal.AddData),ADR('Configuration ID="'));
				brsstrcat(ADR(internal.AddData),ADR(ConfigID));
				brsstrcat(ADR(internal.AddData),ADR('" Configuration version="'));
				brsstrcat(ADR(internal.AddData),ADR(ConfigVersion));
				brsstrcat(ADR(internal.AddData),ADR('"'));
				internal.ArProjectGetInfo_0.Execute := FALSE;
				internal.state := 10;
			ELSIF NOT internal.ArProjectGetInfo_0.Execute THEN
				internal.ArProjectGetInfo_0.Execute := TRUE;
			ELSE
				internal.ArProjectGetInfo_0.Execute := FALSE;
			END_IF;
		10:
			IF internal.ArEventLogGetIdent_0.Done THEN
				internal.ArEventLogGetIdent_0.Execute := FALSE;
				internal.ArEventLogWrite_0.Ident := internal.ArEventLogGetIdent_0.Ident;
				internal.ArEventLogWrite_0.EventID := 1610612736;
				internal.ArEventLogWrite_0.ObjectID := 'HA_Version';
				internal.ArEventLogWrite_0.AddDataFormat := 1;
				internal.ArEventLogWrite_0.AddData := ADR(internal.AddData);
				internal.ArEventLogWrite_0.AddDataSize := brsstrlen(ADR(internal.AddData))+1;
				internal.ArEventLogWrite_0.Execute := TRUE;
				internal.state := 20;
			ELSIF NOT internal.ArEventLogGetIdent_0.Execute THEN
				internal.ArEventLogGetIdent_0.Name := '$$arlogusr';
				internal.ArEventLogGetIdent_0.Execute := TRUE;
			ELSE
				internal.ArEventLogGetIdent_0.Execute := FALSE;
			END_IF;
		20:
			IF internal.ArEventLogWrite_0.Done THEN
				internal.ArEventLogWrite_0.Execute := FALSE;
				internal.state := 30;
			ELSIF NOT internal.ArEventLogWrite_0.Execute THEN
				internal.ArEventLogWrite_0.Execute := TRUE;
			ELSE
				internal.ArEventLogWrite_0.Execute := FALSE;
			END_IF;
		30:
			Done := TRUE;
	END_CASE;

	internal.ArProjectGetInfo_0();
	internal.ArEventLogGetIdent_0();
	internal.ArEventLogWrite_0();

END_FUNCTION_BLOCK
```

### Library Logical/Libraries/HA_Dir (IEC)
Depends on: HA, AsBrStr, standard, brsystem, FileIO, AsUSB, astime

#### Types.typ - Exported data types
```iecst
TYPE
	HA_FileList_typ : 	STRUCT
		Path : STRING[260];
		DateUDINT : UDINT;
		Size : UDINT;
		IsDir : BOOL;
		DirIdx : INT;
		Internal : USINT; (*0=unread, 1=delete, 2=parentDirDelete, 3=remove*)
	END_STRUCT;
	HA_DirDef_typ : 	STRUCT
		Valid : BOOL;
		DirPath : STRING[260];
		Sanitize : HA_DirDef_Sanitize_typ;
	END_STRUCT;
	HA_DirDef_Sanitize_typ : 	STRUCT
		AllowUndefinedDir : BOOL;
		SanitizeFilesByExt : BOOL;
		SanitizeFilesByRoot : BOOL;
		FileExtension : STRING[260];
		FileRoot : STRING[260];
		MaxSize : UDINT;
		MaxFiles : UDINT;
	END_STRUCT;
	HA_DirMake_Internal_typ : 	STRUCT
		State : HA_DIRMAKE_STATE_ENUM;
		DirDefItem : HA_DirDef_typ;
		DirCreate_0 : DirCreate;
		DirIdx : INT;
	END_STRUCT;
	HA_DIRMAKE_STATE_ENUM :
		(
		DIRMAKE_RESET,
		DIRMAKE_IDLE,
		DIRMAKE_CREATE_CMD,
		DIRMAKE_CREATE_WAIT,
		DIRMAKE_DONE,
		DIRMAKE_ERROR
		);
	HA_DirSanitize_Internal_typ : 	STRUCT
		State : HA_DIRSANITIZE_STATE_ENUM;
		DirDeleteEx_0 : DirDeleteEx;
		FileDelete_0 : FileDelete;
		DirDefItem : HA_DirDef_typ;
		FileListItem : HA_FileList_typ;
		FileListItem1 : HA_FileList_typ;
		i : INT;
		j : INT;
		FileListIdx : INT;
		Size : UDINT;
		DirIdent : UDINT;
		SizeCount : UDINT;
		FileCount : UDINT;
		DirData : fiDIR_READ_EX_DATA;
		Found : BOOL;
		Find : INT;
		TempPath : STRING[260];
		CurrentDirIdx : INT;
	END_STRUCT;
	HA_DIRSANITIZE_STATE_ENUM :
		(
		DIRSANITIZE_RESET,
		DIRSANITIZE_IDLE,
		DIRSANITIZE_EVALUATE_DIR,
		DIRSANITIZE_DELETE_DIR_CMD,
		DIRSANITIZE_DELETE_DIR_WAIT,
		DIRSANITIZE_DELETE_DIR_PROCESS,
		DIRSANITIZE_EVALUATE_FILE,
		DIRSANITIZE_DELETE_FILE_CMD,
		DIRSANITIZE_DELETE_FILE_WAIT,
		DIRSANITIZE_DONE,
		DIRSANITIZE_ERROR
		);
	HA_Dir_USB_Connect_Internal_typ : 	STRUCT
		UsbNodeListGet_0 : UsbNodeListGet;
		UsbNodeGet_0 : UsbNodeGet;
		DevLink_0 : DevLink;
		UsbMsDeviceReady_0 : UsbMsDeviceReady;
		DevUnlink_0 : DevUnlink;
		CTON_Delay : CTON;
		NodeList : UDINT;
		Node : usbNode_typ;
		ParString : STRING[1000];
		Handle : UDINT;
		State : HA_USB_CONNECT_STATE_ENUM;
	END_STRUCT;
	HA_USB_CONNECT_STATE_ENUM :
		(
		USB_CONNECT_RESET,
		USB_CONNECT_IDLE,
		USB_CONNECT_GET_LIST_CMD,
		USB_CONNECT_GET_LIST_WAIT,
		USB_CONNECT_GET_NODE_CMD,
		USB_CONNECT_GET_NODE_WAIT,
		USB_CONNECT_DEVLINK_CMD,
		USB_CONNECT_DEVLINK_WAIT,
		USB_CONNECT_CHECK_CONNECTED,
		USB_CONNECT_CONNECTED,
		USB_CONNECT_DEVUNLINK_CMD,
		USB_CONNECT_DEVUNLINK_WAIT,
		USB_CONNECT_DELAY,
		USB_CONNECT_DONE,
		USB_CONNECT_ERROR
		);
	HA_Dir_Transfer_Internal_typ : 	STRUCT
		State : HA_DIR_TRANSFER_STATE_ENUM;
		TransferListItem : HA_Dir_Transfer_List_typ;
		ListIdx : INT;
		DirCopy_0 : DirCopy;
		FileCopy_0 : FileCopy;
		DirDeleteEx_0 : DirDeleteEx;
		DirCreate_0 : DirCreate;
		FileDelete_0 : FileDelete;
	END_STRUCT;
	HA_Dir_Transfer_List_typ : 	STRUCT
		Valid : BOOL;
		SrcOrDestUSB : BOOL;
		IsDir : BOOL;
		SrcDelete : BOOL;
		SrcCreateDir : BOOL;
		NoTransfer : BOOL;
		SrcDev : STRING[80];
		SrcPath : STRING[260];
		DestDev : STRING[80];
		DestPath : STRING[260];
	END_STRUCT;
	HA_DIR_TRANSFER_STATE_ENUM :
		(
		TRANSFER_RESET,
		TRANSFER_IDLE,
		TRANSFER_CHECK_LIST,
		TRANSFER_DIR_COPY_CMD,
		TRANSFER_DIR_COPY_WAIT,
		TRANSFER_FILE_COPY_CMD,
		TRANSFER_FILE_COPY_WAIT,
		TRANSFER_DIR_DELETE_CMD,
		TRANSFER_DIR_DELETE_WAIT,
		TRANSFER_FILE_DELETE_CMD,
		TRANSFER_FILE_DELETE_WAIT,
		TRANSFER_DIR_CREATE_CMD,
		TRANSFER_DIR_CREATE_WAIT,
		TRANSFER_DONE,
		TRANSFER_ERROR
		);
	HA_DirReadAll_Internal_typ : 	STRUCT
		State : HA_DIRREADALL_STATE_ENUM;
		DirOpen_0 : DirOpen;
		DirReadEx_0 : DirReadEx;
		DirClose_0 : DirClose;
		i : INT;
		FileListIdx : INT;
		DirIdent : UDINT;
		DirData : fiDIR_READ_EX_DATA;
		FileListItem : HA_FileList_typ;
		CurrentDirPath : STRING[260];
	END_STRUCT;
	HA_DIRREADALL_STATE_ENUM :
		(
		DIRREADALL_RESET,
		DIRREADALL_IDLE,
		DIRREADALL_OPEN_CMD,
		DIRREADALL_OPEN_WAIT,
		DIRREADALL_READ_CMD,
		DIRREADALL_READ_WAIT,
		DIRREADALL_CLOSE_WAIT,
		DIRREADALL_EVALUATE,
		DIRREADALL_DONE,
		DIRREADALL_ERROR
		);
END_TYPE
```

#### Constants.var - Exported constants
```iecst
VAR CONSTANT
	MAX_DIR_DEF_IDX : INT := 3;
	MAX_DIR_MAN_DELETE_IDX : INT := 99;
	MAX_DIR_MAN_FILE_LIST_IDX : INT := 99;
	MAX_TRANSFER_LIST_IDX : INT := 9;
END_VAR
```

#### HA_Dir.fun - Exported functions and function blocks
```iecst
{REDUND_ERROR} FUNCTION_BLOCK HA_DirMake (* *) (*$GROUP=User,$CAT=User,$GROUPICON=User.png,$CATICON=User.png*)
	VAR_INPUT
		enable : BOOL;
		pDevice : UDINT;
		pDirDef : UDINT;
	END_VAR
	VAR_OUTPUT
		status : UINT;
	END_VAR
	VAR
		Internal : HA_DirMake_Internal_typ;
	END_VAR
END_FUNCTION_BLOCK

{REDUND_ERROR} FUNCTION_BLOCK HA_DirReadAll (*Reads Entire File Device*) (*$GROUP=User,$CAT=User,$GROUPICON=User.png,$CATICON=User.png*)
	VAR_INPUT
		enable : BOOL;
		pDevice : UDINT;
		pFileList : UDINT;
	END_VAR
	VAR_OUTPUT
		status : UINT;
	END_VAR
	VAR
		Internal : HA_DirReadAll_Internal_typ;
	END_VAR
END_FUNCTION_BLOCK

{REDUND_ERROR} FUNCTION_BLOCK HA_DirSanitize (*Sanitizes File Device*) (*$GROUP=User,$CAT=User,$GROUPICON=User.png,$CATICON=User.png*)
	VAR_INPUT
		enable : BOOL;
		pDevice : UDINT;
		pDirDef : UDINT;
		pFileList : UDINT;
	END_VAR
	VAR_OUTPUT
		status : UINT;
	END_VAR
	VAR
		Internal : HA_DirSanitize_Internal_typ;
	END_VAR
END_FUNCTION_BLOCK

{REDUND_ERROR} FUNCTION_BLOCK HA_Dir_USB_Connect (*TODO: Add your comment here*) (*$GROUP=User,$CAT=User,$GROUPICON=User.png,$CATICON=User.png*)
	VAR_INPUT
		enable : BOOL;
		reset : BOOL;
		refresh : BOOL;
		delay : REAL;
	END_VAR
	VAR_OUTPUT
		status : UINT;
		connected : BOOL;
	END_VAR
	VAR
		Internal : HA_Dir_USB_Connect_Internal_typ;
	END_VAR
END_FUNCTION_BLOCK

{REDUND_ERROR} FUNCTION_BLOCK HA_Dir_Transfer (*Transfer List from Device to Another*) (*$GROUP=User,$CAT=User,$GROUPICON=User.png,$CATICON=User.png*)
	VAR_INPUT
		enable : BOOL;
		USB_Connected : BOOL;
		pTransferList : UDINT;
	END_VAR
	VAR_OUTPUT
		index : INT;
		status : UINT;
	END_VAR
	VAR
		Internal : HA_Dir_Transfer_Internal_typ;
	END_VAR
END_FUNCTION_BLOCK
```

#### HA_DirMake.st
```iecst
FUNCTION_BLOCK HA_DirMake

	IF enable = FALSE THEN
		Internal.State									:= DIRMAKE_RESET;
	END_IF;

	CASE Internal.State OF
		DIRMAKE_RESET:
			status										:= 65534;
			brsmemset(ADR(Internal),0,SIZEOF(Internal));
			Internal.State								:= DIRMAKE_IDLE;
		DIRMAKE_IDLE:
			status										:= 65534;
			IF enable THEN
				IF pDevice <> 0 AND pDirDef <> 0 THEN
					status								:= 65535;
					brsmemset(ADR(Internal),0,SIZEOF(Internal));
					Internal.State						:= DIRMAKE_CREATE_CMD;
				ELSE
					status								:= 60001;
					Internal.State						:= DIRMAKE_ERROR;
				END_IF;
			END_IF;
		DIRMAKE_CREATE_CMD:
			status										:= 65535;
			IF Internal.DirIdx >= 0 AND Internal.DirIdx <= MAX_DIR_DEF_IDX THEN
				brsmemcpy(ADR(Internal.DirDefItem),pDirDef+SIZEOF(Internal.DirDefItem)*Internal.DirIdx,SIZEOF(Internal.DirDefItem));
				IF Internal.DirDefItem.Valid THEN
					IF Internal.DirDefItem.DirPath <> '' AND Internal.DirDefItem.DirPath <> '/' THEN
						Internal.DirCreate_0.enable 	:= TRUE;
						Internal.DirCreate_0.pDevice	:= pDevice;
						Internal.DirCreate_0.pName		:= ADR(Internal.DirDefItem.DirPath);
						Internal.State					:= DIRMAKE_CREATE_WAIT;
					ELSE
						Internal.DirIdx 				:= Internal.DirIdx + 1;
					END_IF;
				ELSE
					Internal.State						:= DIRMAKE_DONE;
				END_IF;
			ELSE
				Internal.State							:= DIRMAKE_DONE;
			END_IF;
		DIRMAKE_CREATE_WAIT:
			status										:= 65535;
			IF Internal.DirCreate_0.status = ERR_OK OR Internal.DirCreate_0.status = fiERR_DIR_ALREADY_EXIST THEN
				Internal.DirCreate_0.enable 			:= FALSE;
				Internal.DirIdx 						:= Internal.DirIdx + 1;
				Internal.State 							:= DIRMAKE_CREATE_CMD;
			ELSIF Internal.DirCreate_0.status <> ERR_FUB_BUSY AND Internal.DirCreate_0.status <> ERR_FUB_ENABLE_FALSE THEN
				Internal.DirCreate_0.enable 			:= FALSE;
				status									:= Internal.DirCreate_0.status;
				Internal.State 							:= DIRMAKE_ERROR;
			END_IF;
		DIRMAKE_DONE:
			status										:= 0;
		DIRMAKE_ERROR:
			// Error
	END_CASE;
	Internal.DirCreate_0();

END_FUNCTION_BLOCK
```
